// SIMATIC STEP 7 (V5.x) project Daysil_Autoclav_v4
// CPU: CPU 315-2 PN/DP
// station: P_ADR_BUS
// station: Hardware
// station: SLIO_CPU_015
// program: S7 Program(1)
// program: Backup_11012025
// program: Backup_PID_11012025
// program: Backup_08032025

SYMBOL_TABLE
"AI-SENSOR-DATA"	DB 1	DB 1
"ORTAK_DATA"	DB 2	DB 2	// Ortak Veriler
"TIME_OTO_1_DB"	DB 5	SFB 4
"TIME_OTO_2_DB"	DB 6	SFB 4
"TIME_OTO_1_PROSES_DB"	DB 7	SFB 4
"TIME_OTO_2_PROSES_DB"	DB 8	SFB 4
"SURELER_DB"	DB 14	FB 3
"SAFETY_DB"	DB 15	FB 2
"KAZAN1_DATA"	DB 17	DB 17
"KAZAN2_DATA"	DB 18	DB 18	// KAZAN 2 BILGILERI
"JEN1_DATA"	DB 19	DB 19
"JEN2_DATA"	DB 20	DB 20
"JEN1_PID_DATA"	DB 21	DB 21
"JEN2_PID_DATA"	DB 22	DB 22
"KAZAN1_PID_DATA"	DB 23	DB 23	// KAZAN 1 PID BILGILERI
"KAZAN2_PID_DATA"	DB 24	DB 24	// KAZAN 2 PID BILGILERI
"JEN2_KONTROL_BLOGU_DB"	DB 51	FB 50
"JEN_1_PID_DB"	DB 69	FB 58
"JEN_2_PID_DB"	DB 70	FB 58
"OTOKLAV_1_DB"	DB 94	FB 94
"OTOKLAV_2_DB"	DB 95	FB 95
"FB98_DB"	DB 98	FB 98
"FB99_DB"	DB 99	FB 99
"HMI_DATA"	DB 100	DB 100	// Hmi arayuz verileri
"KAZAN_1_PID_DB"	DB 130	FB 58
"KAZAN_2_PID_DATA"	DB 231	FB 58
"MAINBLOCK"	FB 1	FB 1	// ANA PROGRAM BLOGU
"SAFETY"	FB 2	FB 2
"SURELER"	FB 3	FB 3
"TEST_BLOGU"	FB 5	FB 5
"KAZAN_ORTAK"	FB 20	FB 20
"KAZAN_PID_ORTAK"	FB 21	FB 21
"CONT_C"	FB 41	FB 41	// Continuous Control
"KAZAN_1_PID_KONTROL"	FB 47	FB 47
"KAZAN_2_PID_KONTROL"	FB 48	FB 48
"JEN1_PID_KONTROL"	FB 49	FB 49
"JEN2_PID_KONTROL"	FB 50	FB 50	// BUAHR JENERATÖR 2 PID
"TCONT_CP"	FB 58	FB 58	// temperature PID controller with pulse generator and self-tuning
"KAZAN_1_KONTROL"	FB 94	FB 94
"KAZAN_2_KONTROL"	FB 95	FB 95
"KAZAN1_KONTROL_BLOGU"	FB 96	FB 96
"KAZAN2_KONTROL_BLOGU"	FB 97	FB 97
"JEN1_KONTROL_BLOGU"	FB 98	FB 98
"JEN2_KONTROL_BLOGU"	FB 99	FB 99
"TIME_UNSCALE"	FC 1	FC 1
"O.Vana_AciklikHesaplama"	FC 2	FC 2	// Oransal vana aciklik orani hesaplama
"Int_To_S5Time"	FC 10	FC 10
"Int_To_Second"	FC 11	FC 11
"TIM_S5TI"	FC 40	FC 40	// IEC Time to S5 Time
"SCALE"	FC 105	FC 105	// Scaling Values
"UNSCALE"	FC 106	FC 106	// Unscaling Values
"KAZAN1_ACIL_STOP"	I 0.0	BOOL	// Acil Stop
"KAZAN1_START"	I 0.1	BOOL	// Kazan 1 Start
"KAZAN1_TRANSFER"	I 0.2	BOOL	// Kazan 1 Buhar Transferi
"KAZAN1_BOSALTIM"	I 0.3	BOOL	// Kazan 1 Bosaltim
"KAZAN1_KAPAK_SW"	I 0.4	BOOL	// Kazan 1 Kapak Kapandi
"KAZAN2_ACIL_STOP"	I 0.5	BOOL	// Kazan 2 Acil Stop
"KAZAN2_START"	I 0.6	BOOL	// Kazan 2 Start
"KAZAN2_TRANSFER"	I 0.7	BOOL	// Kazan 2 Buhar Transferi
"KAZAN2_BOSALTIM"	I 1.0	BOOL	// Kazan 2 Bosaltim
"KAZAN2_KAPAK_SW"	I 1.1	BOOL	// Kazan 2 Kapak Kapandi
"JEN1_STOP"	I 1.2	BOOL	// Jenerator 1 Stop
"JEN1_START"	I 1.3	BOOL	// Jenerator 1 Start
"JEN2_STOP"	I 1.4	BOOL	// Jenerator 2 Stop
"JEN2_START"	I 1.5	BOOL	// Jenerator 2 Start
"MANUEL"	I 1.6	BOOL	// Manuel Mod
"OTOMATIK"	I 1.7	BOOL	// Otomatik Mod
"JEN2_MOTOR_CALISTI"	I 2.0	BOOL
"JEN_1_MIN_SU_SEVIYESI"	I 3.0	BOOL
"JEN_2_MIN_SU_SEVIYESI"	I 3.1	BOOL
"0.1 SN."	M 0.0	BOOL
"0.2 SN."	M 0.1	BOOL
"0.4 SN."	M 0.2	BOOL
"0.5 SN."	M 0.3	BOOL
"0.8 SN."	M 0.4	BOOL
"1.0 SN."	M 0.5	BOOL
"1.6 SN."	M 0.6	BOOL
"2.0 SN."	M 0.7	BOOL
"Oto_1_Proses_BASLADI"	M 20.0	BOOL
"Oto_2_Proses_Basladi"	M 20.1	BOOL
"JEN2_CALIS_SURESI_BASLA"	M 22.0	BOOL
"JEN2_CALISTI_RIS"	M 22.1	BOOL
"JEN1_CALIS_SURESI_BASLA"	M 23.0	BOOL
"JEN1_CALISTI_RIS"	M 23.1	BOOL
"Jen1_Guvenlik_set_reset"	M 25.0	BOOL
"Jen2_Guvenlik_Set_Reset"	M 26.0	BOOL
"OTO_1_BEKLEME_BASLADI"	M 27.0	BOOL
"OTO_2_BEKLEME_BASLADI"	M 27.1	BOOL
"KAZAN_1_PID_MAN_ON"	M 35.0	BOOL
"KAZAN_2_MAN_ON"	M 37.0	BOOL
"TEST_START"	M 40.0	BOOL
"TEST_STOP"	M 40.1	BOOL
"TEST_OUT"	M 40.2	BOOL
"ALWAYS OFF"	M 100.0	BOOL	// ALWAYS OFF
"ALWAYS ON"	M 100.1	BOOL	// ALWAYS ON
"SET2_ULASMADI_SR"	M 101.0	BOOL
"SET2_ULASMADI_RIS"	M 101.1	BOOL
"JEN2_TCONT_MAN_ON"	M 155.0	BOOL
"Jen2_Stop_Trigger"	M 200.0	BOOL
"Jen2_Stop_Ris"	M 200.1	BOOL
"Jen2_Stop_Set_Mem"	M 200.2	BOOL
"JEN2_STOP_SET_RESET"	M 201.0	BOOL
"Sicaklik Dustu"	M 201.1	BOOL
"Ris_Jen2_Sicaklik_Dustu"	M 201.2	BOOL
"Rising_Sogutma"	M 201.3	BOOL
"Falling_Sogutma"	M 201.4	BOOL
"JEN1_STOP_SET_RESET"	M 202.0	BOOL
"START"	M 700.1	BOOL
"PID_START"	M 700.2	BOOL
"BRULOR_START"	M 700.3	BOOL
"SICAKLIK_1_OK"	M 700.5	BOOL
"SICAKLIK_2_OK"	M 700.6	BOOL
"BURLOR_MOTOR_START"	M 700.7	BOOL
"STOP"	M 701.1	BOOL
"100_DERECE_RIS"	M 750.0	BOOL
"Jen2_Ris"	M 750.4	BOOL
"Jen1_Ris"	M 750.5	BOOL
"BOS"	M 1000.0	BOOL
"O.VanaIlkAciklik"	MD 42	REAL	// Oransal vana ilk aciklik orani
"O.VanaKademeArtis"	MD 46	REAL	// Oransal vana kademeli artis orani
"PID BLOCK"	OB 35	OB 35	// PID BLOCK
"ZAMANHATASI"	OB 80	OB 80	// ZAMAN HATASI
"GERILIMHATASI"	OB 81	OB 81	// BESLEME GERILIMI HATASI
"HATAUYARISI"	OB 82	OB 82	// HATA UYARISI
"TAKMACIKARMAHATASI"	OB 83	OB 83	// TAKMA ÇIKARMA UYARISI
"CPUHARDWAREERROR"	OB 84	OB 84	// CPU HARDWARE ERROR
"PROGRAMHATASI"	OB 85	OB 85	// PROGRAM YURUTME HATASI
"RACKHATASI"	OB 86	OB 86	// RACK HATASI
"HABERLESMEHATASI"	OB 87	OB 87	// HABERLESME HATASI,
"COMPLETE RESTART"	OB 100	OB 100	// Complete Restart
"RESTART"	OB 101	OB 101	// Restart
"COLD RESTART"	OB 102	OB 102	// Cold Restart
"PROGRAMMINGERROR"	OB 121	OB 121	// PROGRAMLAMA HATASI
"MOD_ERR"	OB 122	OB 122	// Module Access Error
"KAZAN1_YESIL_LAMBA"	Q 0.0	BOOL	// Kazan 1 Yesil Lamba
"KAZAN1_KIRMIZI_LAMBA"	Q 0.1	BOOL	// Kazan 1 Kirmizi Lamba
"KAZAN1_DUDUK"	Q 0.2	BOOL	// Kazan 1 Duduk
"KAZAN1_BOSALTIM_VALFI"	Q 0.3	BOOL	// Kazan 1 Buhar Bosaltim
"KAZAN1_TRANS_BUT_LAMBASI"	Q 0.4	BOOL	// Kazan 1 Transfer Lambasi
"KAZAN1_EMN_VALFI_BOS"	Q 0.5	BOOL	// Kazan  1 Emniyet vantili bosaltim valfi
"KAZAN2_YESIL_LAMBA"	Q 0.6	BOOL	// Kazan 2 Yesil Lamba
"KAZAN2_KIRMIZI_LAMBA"	Q 0.7	BOOL	// Kazan 2 Kirmizi Lamba
"KAZAN2_DUDUK"	Q 1.0	BOOL	// Kazan 2 Duduk
"KAZAN2_BOSALTIM_VALFI"	Q 1.1	BOOL	// Kazan 2 Buhar Bosaltim
"KAZAN2_TRANS_BUT_LAMBASI"	Q 1.2	BOOL	// Kazan 2 Transfer Lambasi
"KAZAN2_EMN_VALFI_BOS"	Q 1.3	BOOL	// Kazan Emniyet vantili bosaltim valfi
"JEN_1_HAT_VANASI"	Q 1.4	BOOL
"JEN_1_PANO_STOP_LAMBASI"	Q 1.5	BOOL
"JEN_1_PANO_START_LAMBASI"	Q 1.6	BOOL
"JEN_2_HAT_VANASI"	Q 1.7	BOOL
"JEN_2_PANO_STOP_LAMBASI"	Q 2.0	BOOL
"JEN_2_PANO_START_LAMBASI"	Q 2.1	BOOL
"PANO_OTO_MAN_BUTON_LAMBA"	Q 2.2	BOOL
"PANO_ALARM"	Q 2.3	BOOL
"JEN_1_BRULOR"	Q 2.4	BOOL
"JEN_1_POMPA"	Q 2.5	BOOL
"JEN_2_BRULOR_OUT"	Q 2.6	BOOL
"JEN_2_SU_POM_OUT"	Q 2.7	BOOL
"TON"	SFB 4	SFB 4	// Generate an On Delay
"TIME_TCK"	SFC 64	SFC 64	// Read the System Time
"delay_300ms_1"	T 8	TIMER
"500ms_delay1"	T 10	TIMER
"1s Delay"	T 11	TIMER
"Pisim_Suresi"	T 12	TIMER
"500ms_delay"	T 13	TIMER
"s_offt_7s_delay"	T 14	TIMER
"tm_adim1_pid_basla_delay"	T 16	TIMER
"500ms_delay_kazan_2"	T 20	TIMER
"1ms_delay_kazan_2"	T 21	TIMER
"kazan_2_pisirme_delay"	T 22	TIMER
"kazan_2_500ms_delay"	T 23	TIMER
"kazan_2_7s_delay"	T 24	TIMER
"Delay_500ms_Jen2"	T 30	TIMER
"DELAY_1S_JEN_HATA"	T 33	TIMER
"DELAY_300MS"	T 42	TIMER
"DELAY_500MS_1"	T 43	TIMER
"DELAY_5S_pompa"	T 44	TIMER
"OTO_2_DELAY_BITIS"	T 50	TIMER
"OTO_1_DELAY_PISIM_BITTI"	T 51	TIMER
"DELAY_ADIM5_BEKLE"	T 52	TIMER
"DELAY_ADIM5_BEKLE2"	T 53	TIMER
"TIM_SET2_ULASMADI"	T 57	TIMER
"VAT_1"	VAT 1	
END_SYMBOL_TABLE

FUNCTION_BLOCK "MAINBLOCK"	// FB 1
VERSION : 0.1
BEGIN
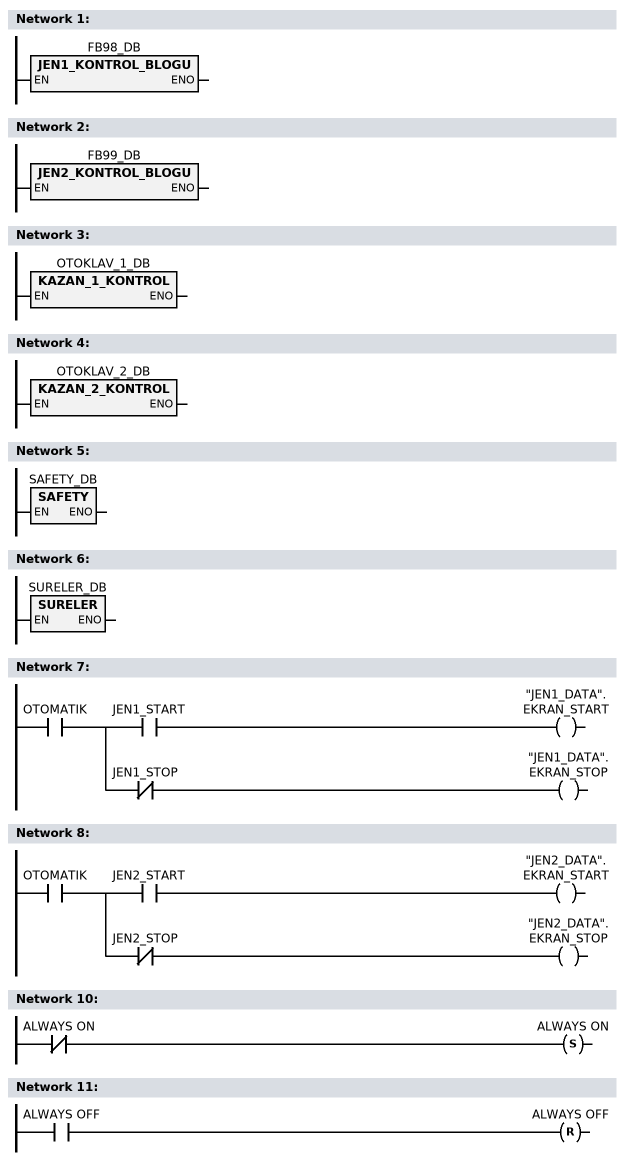
NETWORK
TITLE =
      CALL  "JEN1_KONTROL_BLOGU" , "FB98_DB";
      NOP   0;
NETWORK
TITLE =
      CALL  "JEN2_KONTROL_BLOGU" , "FB99_DB";
      NOP   0;
NETWORK
TITLE =
      CALL  "KAZAN_1_KONTROL" , "OTOKLAV_1_DB";
      NOP   0;
NETWORK
TITLE =
      CALL  "KAZAN_2_KONTROL" , "OTOKLAV_2_DB";
      NOP   0;
NETWORK
TITLE =
      CALL  "SAFETY" , "SAFETY_DB";
      NOP   0;
NETWORK
TITLE =
      CALL  "SURELER" , "SURELER_DB";
      NOP   0;
NETWORK
TITLE =
      A     "OTOMATIK";
      =     L 0.0;
      A     L 0.0;
      A     "JEN1_START";
      =     "JEN1_DATA".EKRAN_START;
      A     L 0.0;
      AN    "JEN1_STOP";
      =     "JEN1_DATA".EKRAN_STOP;
NETWORK
TITLE =
      A     "OTOMATIK";
      =     L 0.0;
      A     L 0.0;
      A     "JEN2_START";
      =     "JEN2_DATA".EKRAN_START;
      A     L 0.0;
      AN    "JEN2_STOP";
      =     "JEN2_DATA".EKRAN_STOP;
NETWORK
TITLE =
NETWORK
TITLE =
      AN    "ALWAYS ON";
      S     "ALWAYS ON";
NETWORK
TITLE =
      A     "ALWAYS OFF";
      R     "ALWAYS OFF";
NETWORK
TITLE =
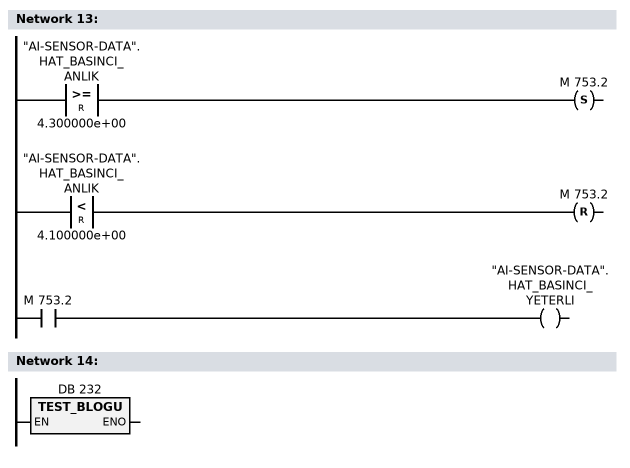
NETWORK
TITLE =
      A(;
      L     "AI-SENSOR-DATA".HAT_BASINCI_ANLIK;
      L     4.300000e+00;
      >=R;
      );
      S     M 753.2;
      A(;
      L     "AI-SENSOR-DATA".HAT_BASINCI_ANLIK;
      L     4.100000e+00;
      <R;
      );
      R     M 753.2;
      A     M 753.2;
      =     "AI-SENSOR-DATA".HAT_BASINCI_YETERLI;
NETWORK
TITLE =
      CALL  "TEST_BLOGU" , DB 232;
      NOP   0;
END_FUNCTION_BLOCK

FUNCTION_BLOCK "SAFETY"	// FB 2
VERSION : 0.1
BEGIN
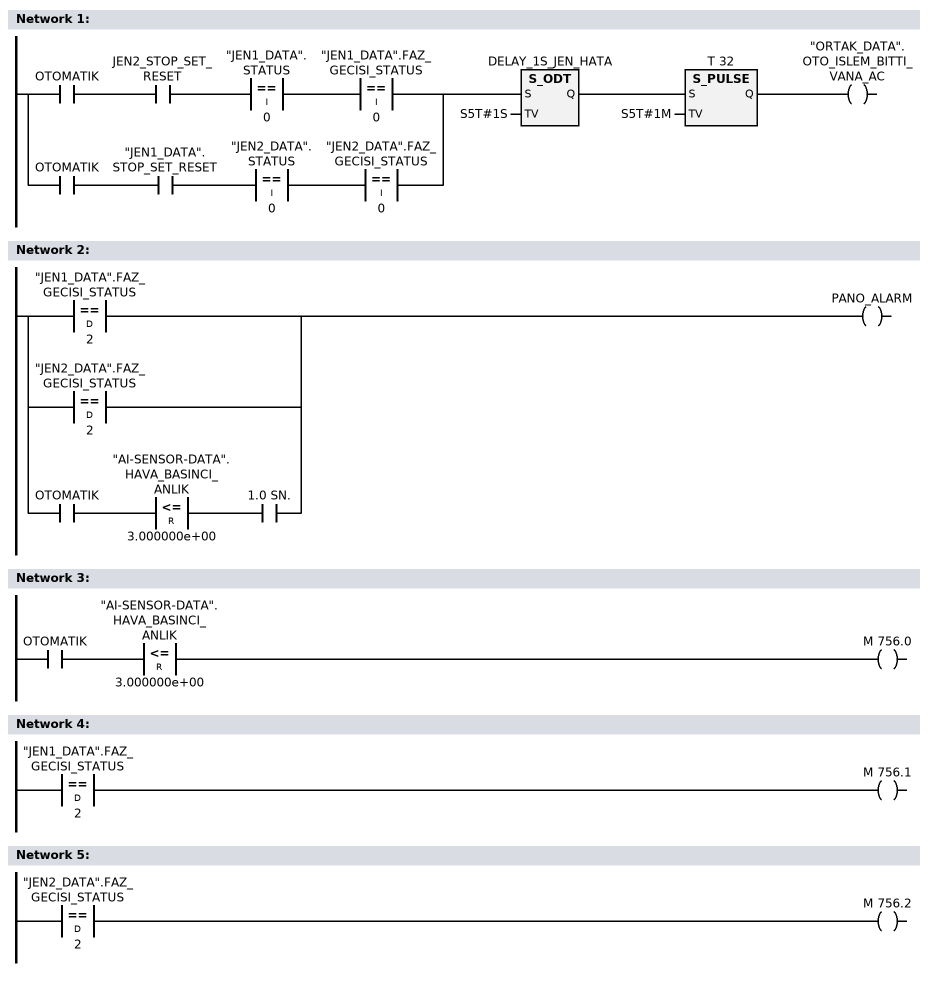
NETWORK
TITLE =
      A(;
      A(;
      A     "OTOMATIK";
      A     "JEN2_STOP_SET_RESET";
      A(;
      L     "JEN1_DATA".STATUS;
      L     0;
      ==I;
      );
      A(;
      L     "JEN1_DATA".FAZ_GECISI_STATUS;
      L     0;
      ==I;
      );
      O;
      A     "OTOMATIK";
      A     "JEN1_DATA".STOP_SET_RESET;
      A(;
      L     "JEN2_DATA".STATUS;
      L     0;
      ==I;
      );
      A(;
      L     "JEN2_DATA".FAZ_GECISI_STATUS;
      L     0;
      ==I;
      );
      );
      L     S5T#1S;
      SD    "DELAY_1S_JEN_HATA";
      NOP   0;
      NOP   0;
      NOP   0;
      A     "DELAY_1S_JEN_HATA";
      );
      L     S5T#1M;
      SP    T 32;
      NOP   0;
      NOP   0;
      NOP   0;
      A     T 32;
      =     "ORTAK_DATA".OTO_ISLEM_BITTI_VANA_AC;
NETWORK
TITLE =
      O(;
      L     "JEN1_DATA".FAZ_GECISI_STATUS;
      L     2;
      ==D;
      );
      O(;
      L     "JEN2_DATA".FAZ_GECISI_STATUS;
      L     2;
      ==D;
      );
      O;
      A     "OTOMATIK";
      A(;
      L     "AI-SENSOR-DATA".HAVA_BASINCI_ANLIK;
      L     3.000000e+00;
      <=R;
      );
      A     "1.0 SN.";
      =     "PANO_ALARM";
NETWORK
TITLE =
      A     "OTOMATIK";
      A(;
      L     "AI-SENSOR-DATA".HAVA_BASINCI_ANLIK;
      L     3.000000e+00;
      <=R;
      );
      =     M 756.0;
NETWORK
TITLE =
      L     "JEN1_DATA".FAZ_GECISI_STATUS;
      L     2;
      ==D;
      =     M 756.1;
NETWORK
TITLE =
      L     "JEN2_DATA".FAZ_GECISI_STATUS;
      L     2;
      ==D;
      =     M 756.2;
END_FUNCTION_BLOCK

FUNCTION_BLOCK "SURELER"	// FB 3
VERSION : 0.1
BEGIN
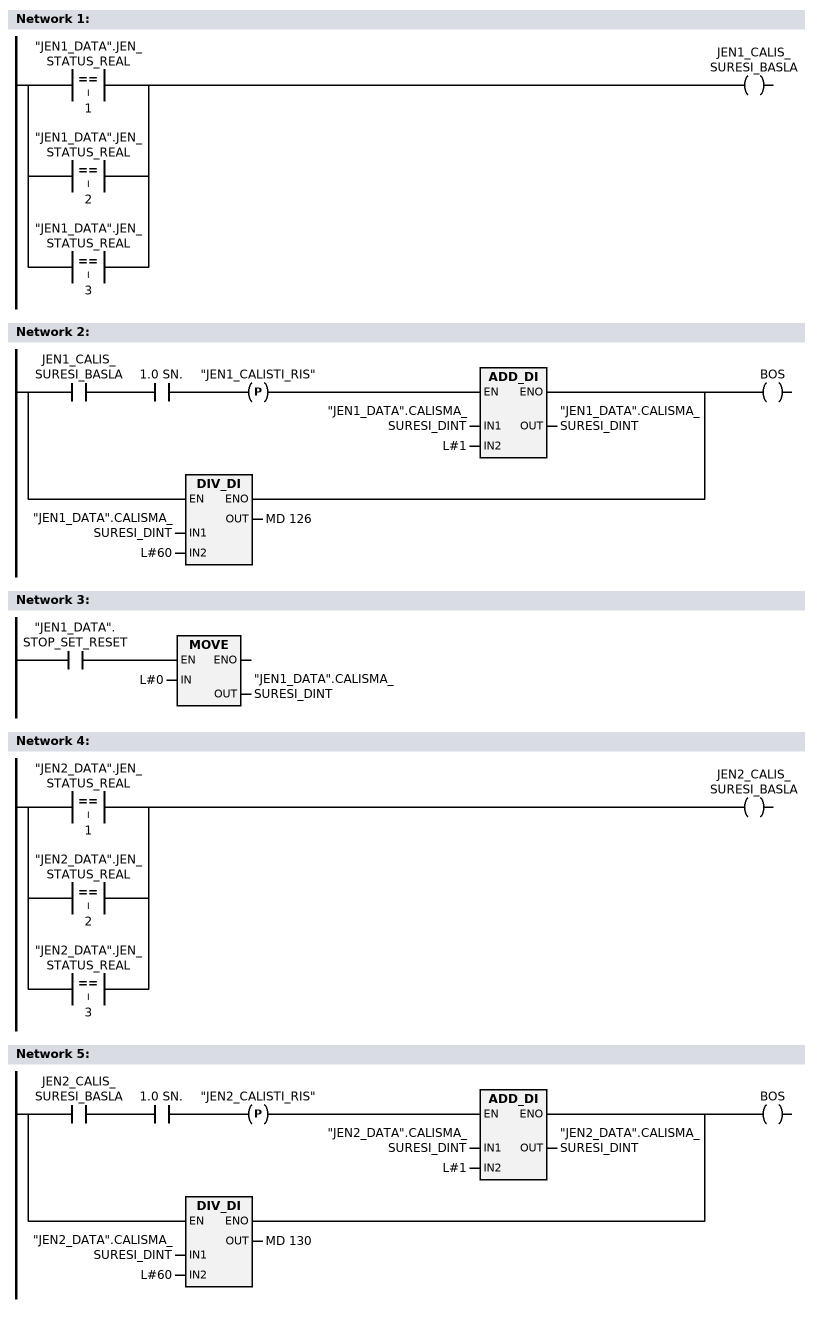
NETWORK
TITLE =
      O(;
      L     "JEN1_DATA".JEN_STATUS_REAL;
      L     1;
      ==I;
      );
      O(;
      L     "JEN1_DATA".JEN_STATUS_REAL;
      L     2;
      ==I;
      );
      O(;
      L     "JEN1_DATA".JEN_STATUS_REAL;
      L     3;
      ==I;
      );
      =     "JEN1_CALIS_SURESI_BASLA";
NETWORK
TITLE =
      O(;
      A     "JEN1_CALIS_SURESI_BASLA";
      A     "1.0 SN.";
      FP    "JEN1_CALISTI_RIS";
      JNB   _001;
      L     "JEN1_DATA".CALISMA_SURESI_DINT;
      L     L#1;
      +D;
      T     "JEN1_DATA".CALISMA_SURESI_DINT;
      AN    OV;
      SAVE;
      CLR;
_001: A     BR;
      );
      O(;
      L     "JEN1_DATA".CALISMA_SURESI_DINT;
      L     L#60;
      /D;
      T     MD 126;
      AN    OV;
      SAVE;
      CLR;
      A     BR;
      );
      =     "BOS";
NETWORK
TITLE =
      A     "JEN1_DATA".STOP_SET_RESET;
      JNB   _002;
      L     L#0;
      T     "JEN1_DATA".CALISMA_SURESI_DINT;
_002: NOP   0;
NETWORK
TITLE =
      O(;
      L     "JEN2_DATA".JEN_STATUS_REAL;
      L     1;
      ==I;
      );
      O(;
      L     "JEN2_DATA".JEN_STATUS_REAL;
      L     2;
      ==I;
      );
      O(;
      L     "JEN2_DATA".JEN_STATUS_REAL;
      L     3;
      ==I;
      );
      =     "JEN2_CALIS_SURESI_BASLA";
NETWORK
TITLE =
      O(;
      A     "JEN2_CALIS_SURESI_BASLA";
      A     "1.0 SN.";
      FP    "JEN2_CALISTI_RIS";
      JNB   _003;
      L     "JEN2_DATA".CALISMA_SURESI_DINT;
      L     L#1;
      +D;
      T     "JEN2_DATA".CALISMA_SURESI_DINT;
      AN    OV;
      SAVE;
      CLR;
_003: A     BR;
      );
      O(;
      L     "JEN2_DATA".CALISMA_SURESI_DINT;
      L     L#60;
      /D;
      T     MD 130;
      AN    OV;
      SAVE;
      CLR;
      A     BR;
      );
      =     "BOS";
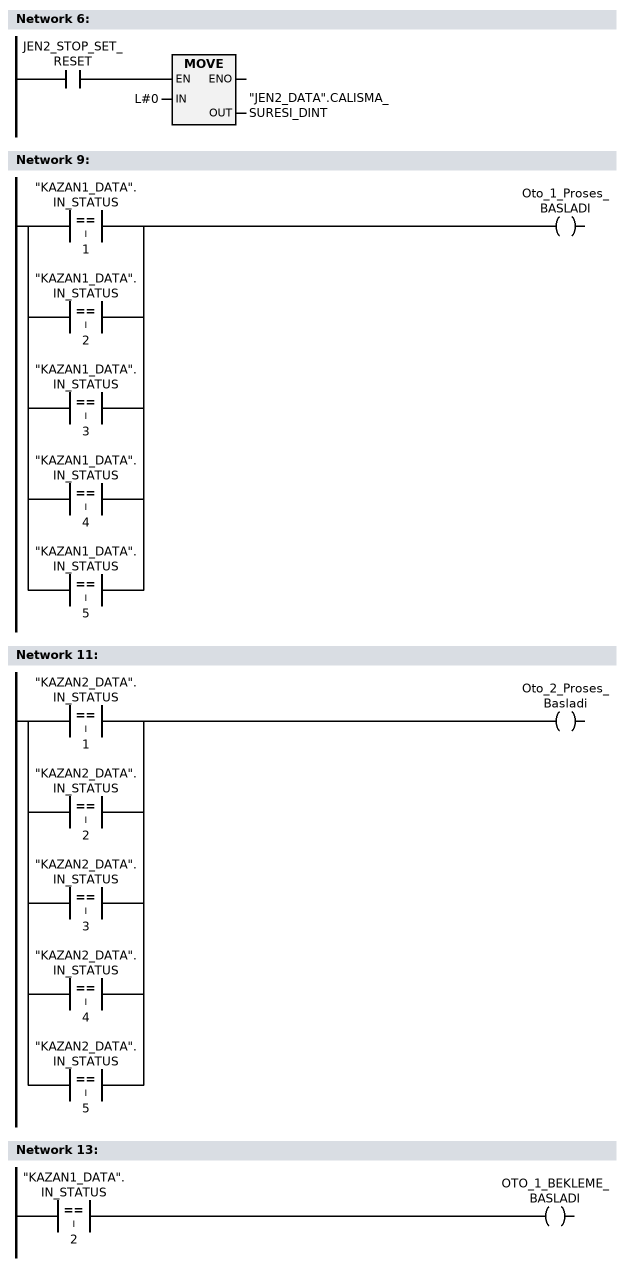
NETWORK
TITLE =
      A     "JEN2_STOP_SET_RESET";
      JNB   _004;
      L     L#0;
      T     "JEN2_DATA".CALISMA_SURESI_DINT;
_004: NOP   0;
NETWORK
TITLE =
      O(;
      A(;
      A     "KAZAN1_DATA".O_PISIM_BASLADI;
      =     L 0.0;
      BLD   103;
      BLD   9;
      =     L 5.0;
      CDB;
      OPN   DI 5;
      TAR2  LD 1;
      A     L 0.0;
      =     DIX 0.0;
      L     L#82800000;
      T     DID 2;
      LAR2  P#DBX 0.0;
      UC    "TON";
      LAR2  LD 1;
      L     DID 8;
      OPN   DI 17;
      T     DID 42;
      OPN   DI 5;
      CDB;
      BLD   10;
      A     BR;
      );
      JNB   _005;
      CALL  "TIME_UNSCALE" (
           $1                       := "KAZAN1_DATA".PISIM_GECEN_SURE_TIME,
           $2                       := "KAZAN1_DATA".IN_PISIM_SURESI,
           $3                       := "KAZAN1_DATA".PISIM_GECEN_SURE_DINT);
_005: A     BR;
      );
      O(;
      L     "KAZAN1_DATA".PISIM_GECEN_SURE_DINT;
      L     60;
      /D;
      T     MD 118;
      AN    OV;
      SAVE;
      CLR;
      A     BR;
      );
      =     "BOS";
NETWORK
TITLE =
      O(;
      A(;
      A     "KAZAN2_DATA".O_PISIM_BASLADI;
      =     L 0.0;
      BLD   103;
      BLD   9;
      =     L 5.0;
      CDB;
      OPN   DI 6;
      TAR2  LD 1;
      A     L 0.0;
      =     DIX 0.0;
      L     L#82800000;
      T     DID 2;
      LAR2  P#DBX 0.0;
      UC    "TON";
      LAR2  LD 1;
      L     DID 8;
      OPN   DI 18;
      T     DID 42;
      OPN   DI 6;
      CDB;
      BLD   10;
      A     BR;
      );
      JNB   _006;
      CALL  "TIME_UNSCALE" (
           $1                       := "KAZAN2_DATA".PISIM_GECEN_SURE_TIME,
           $2                       := "KAZAN2_DATA".IN_PISIM_SURESI,
           $3                       := "KAZAN2_DATA".PISIM_GECEN_SURE_DINT);
_006: A     BR;
      );
      O(;
      L     "KAZAN2_DATA".PISIM_GECEN_SURE_DINT;
      L     60;
      /D;
      T     MD 122;
      AN    OV;
      SAVE;
      CLR;
      A     BR;
      );
      =     "BOS";
NETWORK
TITLE =
      O(;
      L     "KAZAN1_DATA".IN_STATUS;
      L     1;
      ==I;
      );
      O(;
      L     "KAZAN1_DATA".IN_STATUS;
      L     2;
      ==I;
      );
      O(;
      L     "KAZAN1_DATA".IN_STATUS;
      L     3;
      ==I;
      );
      O(;
      L     "KAZAN1_DATA".IN_STATUS;
      L     4;
      ==I;
      );
      O(;
      L     "KAZAN1_DATA".IN_STATUS;
      L     5;
      ==I;
      );
      =     "Oto_1_Proses_BASLADI";
NETWORK
TITLE =
      O(;
      A(;
      A     "Oto_1_Proses_BASLADI";
      =     L 0.0;
      BLD   103;
      BLD   9;
      =     L 5.0;
      CDB;
      OPN   DI 7;
      TAR2  LD 1;
      A     L 0.0;
      =     DIX 0.0;
      L     L#82800000;
      T     DID 2;
      LAR2  P#DBX 0.0;
      UC    "TON";
      LAR2  LD 1;
      L     DID 8;
      OPN   DI 17;
      T     DID 50;
      OPN   DI 7;
      CDB;
      BLD   10;
      A     BR;
      );
      JNB   _007;
      L     "KAZAN1_DATA".PROSES_SURESI_TIME;
      L     1000;
      /D;
      T     "KAZAN1_DATA".PROSES_SURESI_DINT;
      AN    OV;
      SAVE;
      CLR;
_007: A     BR;
      );
      O(;
      L     "KAZAN1_DATA".PROSES_SURESI_DINT;
      L     60;
      /D;
      T     MD 110;
      AN    OV;
      SAVE;
      CLR;
      A     BR;
      );
      =     "BOS";
NETWORK
TITLE =
      O(;
      L     "KAZAN2_DATA".IN_STATUS;
      L     1;
      ==I;
      );
      O(;
      L     "KAZAN2_DATA".IN_STATUS;
      L     2;
      ==I;
      );
      O(;
      L     "KAZAN2_DATA".IN_STATUS;
      L     3;
      ==I;
      );
      O(;
      L     "KAZAN2_DATA".IN_STATUS;
      L     4;
      ==I;
      );
      O(;
      L     "KAZAN2_DATA".IN_STATUS;
      L     5;
      ==I;
      );
      =     "Oto_2_Proses_Basladi";
NETWORK
TITLE =
      O(;
      A(;
      A     "Oto_2_Proses_Basladi";
      =     L 0.0;
      BLD   103;
      BLD   9;
      =     L 5.0;
      CDB;
      OPN   DI 8;
      TAR2  LD 1;
      A     L 0.0;
      =     DIX 0.0;
      L     L#82800000;
      T     DID 2;
      LAR2  P#DBX 0.0;
      UC    "TON";
      LAR2  LD 1;
      L     DID 8;
      OPN   DI 18;
      T     DID 50;
      OPN   DI 8;
      CDB;
      BLD   10;
      A     BR;
      );
      JNB   _008;
      L     "KAZAN2_DATA".PROSES_SURESI_TIM;
      L     1000;
      /D;
      T     "KAZAN2_DATA".PROSES_SURESI_DINT;
      AN    OV;
      SAVE;
      CLR;
_008: A     BR;
      );
      O(;
      L     "KAZAN2_DATA".PROSES_SURESI_DINT;
      L     60;
      /D;
      T     MD 114;
      AN    OV;
      SAVE;
      CLR;
      A     BR;
      );
      =     "BOS";
NETWORK
TITLE =
      L     "KAZAN1_DATA".IN_STATUS;
      L     2;
      ==I;
      =     "OTO_1_BEKLEME_BASLADI";
NETWORK
TITLE =
      A(;
      A     "OTO_1_BEKLEME_BASLADI";
      =     L 0.0;
      BLD   103;
      BLD   9;
      =     L 5.0;
      CDB;
      OPN   DI 9;
      TAR2  LD 1;
      A     L 0.0;
      =     DIX 0.0;
      L     L#82800000;
      T     DID 2;
      LAR2  P#DBX 0.0;
      UC    "TON";
      LAR2  LD 1;
      L     DID 8;
      OPN   DI 17;
      T     DID 58;
      OPN   DI 9;
      CDB;
      BLD   10;
      A     BR;
      );
      JNB   _009;
      L     "KAZAN1_DATA".BEKLEME_SURESI_TIME;
      L     1000;
      /D;
      T     "KAZAN1_DATA".BEKLEME_SURESI_DINT;
_009: NOP   0;
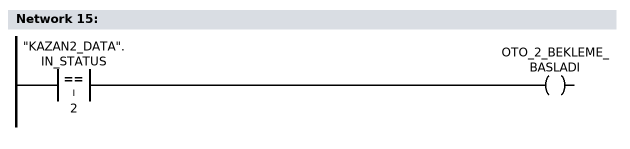
NETWORK
TITLE =
      L     "KAZAN2_DATA".IN_STATUS;
      L     2;
      ==I;
      =     "OTO_2_BEKLEME_BASLADI";
NETWORK
TITLE =
      A(;
      A     "OTO_2_BEKLEME_BASLADI";
      =     L 0.0;
      BLD   103;
      BLD   9;
      =     L 5.0;
      CDB;
      OPN   DI 10;
      TAR2  LD 1;
      A     L 0.0;
      =     DIX 0.0;
      L     L#82800000;
      T     DID 2;
      LAR2  P#DBX 0.0;
      UC    "TON";
      LAR2  LD 1;
      L     DID 8;
      OPN   DI 18;
      T     DID 58;
      OPN   DI 10;
      CDB;
      BLD   10;
      A     BR;
      );
      JNB   _00a;
      L     "KAZAN2_DATA".BEKLEME_SURESI_TIME;
      L     1000;
      /D;
      T     "KAZAN2_DATA".BEKLEME_SURESI_DINT;
_00a: NOP   0;
END_FUNCTION_BLOCK

FUNCTION_BLOCK "TEST_BLOGU"	// FB 5
VERSION : 0.1
BEGIN
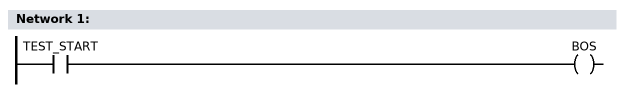
NETWORK
TITLE =
      A     "TEST_START";
      =     "BOS";
END_FUNCTION_BLOCK

FUNCTION_BLOCK "KAZAN_ORTAK"	// FB 20
VERSION : 0.1
VAR_INPUT
  IN_ACIL_STOP : BOOL ;
  IN_START : BOOL ;
  IN_TRANSFER : BOOL ;
  IN_BOSALTIM : BOOL ;
  IN_KAPAK : BOOL ;
  IN_JEN1_OK : BOOL ;
  IN_JEN2_OK : BOOL ;
  IN_JENS_OK : BOOL ;
  IN_TRANSFERE_HAZIR : BOOL ;
  IN_PISIM_SURESI : S5TIME ;
  IN_SCALE_BASINC_PER : INT ;
  IN_SET_BASINC : REAL ;
  IN_DIGER_KAZAN_BASINCI : REAL ;
  IN_TIMER_500MS : TIMER ;
  IN_TIMER_1S : TIMER ;
  IN_TIMER_PISIRME : TIMER ;
  IN_TIMER_500MS_2 : TIMER ;
  IN_TIMER_7S : TIMER ;
  IN_SCALE_HI_LIM : REAL ;
  IN_SCALE_LO_LIM : REAL ;
  IN_SCALE_SICAKLIK_HI_LIM : REAL ;
  IN_SCALE_SICAKLIK_LO_LIM : REAL ;
  IN_SCALE_SICAKLIK_PER : INT ;
  IN_DIGER_KAZAN_BOSALTIMD : BOOL ;
  IN_TRANSFER_BASLADI : BOOL ;
  IN_PISIM_SURESI_TIME_DB : BLOCK_DB ;
  IN_DIG_KAZAN_PROSES_BAS : BOOL ;
  IN_JEN_DURDU : BOOL ;
  IN_JEN_DURDUR_PID_MAN : REAL ;
  IN_DELAY_BITISI_BEKLE : TIMER ;
  IN_DELAY_BIRAZ_BEKLE : TIMER ;
  IN31 : TIMER ;
  IN32 : TIMER ;
  Bos_Vana_Period_Timer : TIMER ;
  Bos_Vana_Aciklik_Timer : TIMER ;
  BosVana_Per_TimeInterval : INT ;	//Bosaltim vanasi periyod timer interval degeri
  BosVana_Aci_TimeInterval : INT ;	//Bosaltim vanasi aciklik timer interval degeri
  BosVana_Acik_Sayisi : INT ;	//Bosaltim valfi acik kalma tekrar sayisi
END_VAR
VAR_OUTPUT
  O_YESIL_LAM : BOOL ;
  O_KIRMIZI_LAM : BOOL ;
  O_DUDUK : BOOL ;
  O_BOSALTIM_VALFI : BOOL ;
  O_PID_MAN_ON : BOOL ;
  O_PID_MAN : REAL ;
  O_TRANSFER_YAPILIYOR : BOOL ;
  O_SCALE_BASINC_RET_VAL : WORD ;
  O_SCALE_BASINC_OUT : REAL ;
  O_EMNIYET_VALFI : BOOL ;
  O_TRANSFERE_HAZIR : BOOL ;
  O_SCALE_SICAKLIK_RET_VAL : WORD ;
  O_SCALE_SICAKLIK_OUT : REAL ;
  O_TRANSFER_ET_LAMBASI : BOOL ;
  O_PROSES_BASLADI : BOOL ;
  O_KAZAN_BOSALTIMDA : BOOL ;
  O_PISIM_BASLADI : BOOL ;
END_VAR
VAR_IN_OUT
  STATUS : INT ;
END_VAR
VAR
  ST_STATUS : INT ;
  ST_OUT_BOSALTIM_MEM : BOOL ;
  ST_OUT_PID_MAN_ON : BOOL ;
  ST_OUT_PID_MAN : REAL ;
  st_ris_pid_zero : BOOL ;
  st_scale_hi_lim : REAL  := 1.000000e+001;
  st_scale_lo_lim : REAL ;
  st_basinc_ok_sure_basla : BOOL ;
  st_tolerans_mul : REAL ;
  st_toleransli_basinc : REAL ;
  st_adim4_bosaltim_valfi : BOOL ;
  st_OUT_adim4_emnyet_val : BOOL ;
  st_pid_basla : BOOL ;
  st_bosalti_valfi_acil : BOOL ;
  st_scale_basinc_ret_val : WORD ;
  st_scale_basinc_out : REAL ;
  st_scale_sicaklik_ret_va : WORD ;
  st_scale_sicaklik_out : REAL ;
  ST_PROSES_BASLADI : BOOL ;
  ST_KAZAN_BOSALTIMDA : BOOL ;
  ST_BOS : BOOL ;
  ST_SET_ADD_BASINC_02 : REAL ;
  ST_GECEN_PISIM_SURESI : TIME ;
  st_5_bar_ustu : BOOL ;
  st_5_bar_alti : BOOL ;
  st_5_bar_guvenlik_SR : BOOL ;
  st_5_bar_guvenlik_mem : BOOL ;
  STAT78 : BOOL ;
  stBasVana_Per_TimeIn : S5TIME ;
  stBasVana_Aci_TimeIn : S5TIME ;
  stBasVana_Aci_Ris : BOOL ;
  stBasVana_Aci_Sayisi : INT ;
  stBosVanasini_Ac : BOOL ;
END_VAR
VAR_TEMP
  tKademe : STRUCT
   Bir : REAL ;
   Iki : REAL ;
   Uc : REAL ;
   Dort : REAL ;
   Bes : REAL ;
   Alti : REAL ;
   Yedi : REAL ;
  END_STRUCT ;
END_VAR
BEGIN
NETWORK
TITLE = BASLANGIC SARTLARI
      A(;
      A(;
      A     "ALWAYS OFF";
      =     L 28.0;
      BLD   103;
      CALL  "SCALE" (
           $1                       := #IN_SCALE_BASINC_PER,
           $2                       := #IN_SCALE_HI_LIM,
           $3                       := #IN_SCALE_LO_LIM,
           $4                       := L 28.0,
           $5                       := #st_scale_basinc_ret_val,
           $6                       := #st_scale_basinc_out);
      A     BR;
      );
      JNB   _001;
      L     #st_scale_basinc_ret_val;
      T     #O_SCALE_BASINC_RET_VAL;
      SET;
      SAVE;
      CLR;
_001: A     BR;
      );
      JNB   _002;
      L     #st_scale_basinc_out;
      T     #O_SCALE_BASINC_OUT;
_002: NOP   0;
NETWORK
TITLE =
      A(;
      A(;
      A     "ALWAYS OFF";
      =     L 28.0;
      BLD   103;
      CALL  "SCALE" (
           $1                       := #IN_SCALE_SICAKLIK_PER,
           $2                       := #IN_SCALE_SICAKLIK_HI_LIM,
           $3                       := #IN_SCALE_SICAKLIK_LO_LIM,
           $4                       := L 28.0,
           $5                       := #st_scale_sicaklik_ret_va,
           $6                       := #st_scale_sicaklik_out);
      A     BR;
      );
      JNB   _003;
      L     #st_scale_sicaklik_ret_va;
      T     #O_SCALE_SICAKLIK_RET_VAL;
      SET;
      SAVE;
      CLR;
_003: A     BR;
      );
      JNB   _004;
      L     #st_scale_sicaklik_out;
      T     #O_SCALE_SICAKLIK_OUT;
_004: NOP   0;
NETWORK
TITLE = START
      A(;
      A     "OTOMATIK";
      A     #IN_ACIL_STOP;
      A     "AI-SENSOR-DATA".HAT_BASINCI_YETERLI;
      L     S5T#200MS;
      T     LD 28;
      TAK;
      T     LD 32;
      L     #IN_TIMER_500MS;
      T     LW 36;
      L     LD 32;
      L     LD 28;
      SD    T [LW 36];
      NOP   0;
      NOP   0;
      NOP   0;
      T     LD 28;
      TAK;
      T     LD 32;
      L     #IN_TIMER_500MS;
      T     LW 36;
      L     LD 32;
      L     LD 28;
      A     T [LW 36];
      );
      A     #IN_KAPAK;
      A     #IN_START;
      A(;
      L     #STATUS;
      L     0;
      ==I;
      );
      JNB   _005;
      L     1;
      T     #STATUS;
      SET;
      SAVE;
      CLR;
_005: A     BR;
      S     #ST_PROSES_BASLADI;
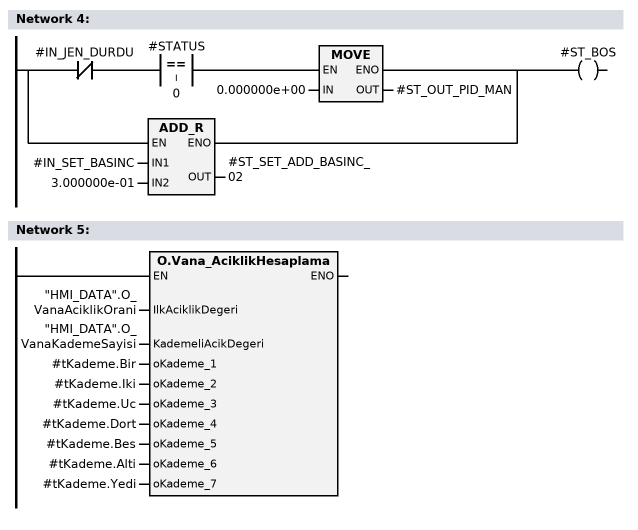
NETWORK
TITLE =
//1-Baslangicta vakum olmamasi icin bosaltim valfini ac
//Valf Normalde acik gibi dusundum
//2-Oransal valfi kapali tut
      O(;
      AN    #IN_JEN_DURDU;
      A(;
      L     #STATUS;
      L     0;
      ==I;
      );
      JNB   _006;
      L     0.000000e+00;
      T     #ST_OUT_PID_MAN;
      SET;
      SAVE;
      CLR;
_006: A     BR;
      );
      O(;
      L     #IN_SET_BASINC;
      L     3.000000e-01;
      +R;
      T     #ST_SET_ADD_BASINC_02;
      AN    OV;
      SAVE;
      CLR;
      A     BR;
      );
      =     #ST_BOS;
NETWORK
TITLE =
      CALL  "O.Vana_AciklikHesaplama" (
           IlkAciklikDegeri         := "HMI_DATA".O_VanaAciklikOrani,
           KademeliAcikDegeri       := "HMI_DATA".O_VanaKademeSayisi,
           oKademe_1                := #tKademe.Bir,
           oKademe_2                := #tKademe.Iki,
           oKademe_3                := #tKademe.Uc,
           oKademe_4                := #tKademe.Dort,
           oKademe_5                := #tKademe.Bes,
           oKademe_6                := #tKademe.Alti,
           oKademe_7                := #tKademe.Yedi);
      NOP   0;
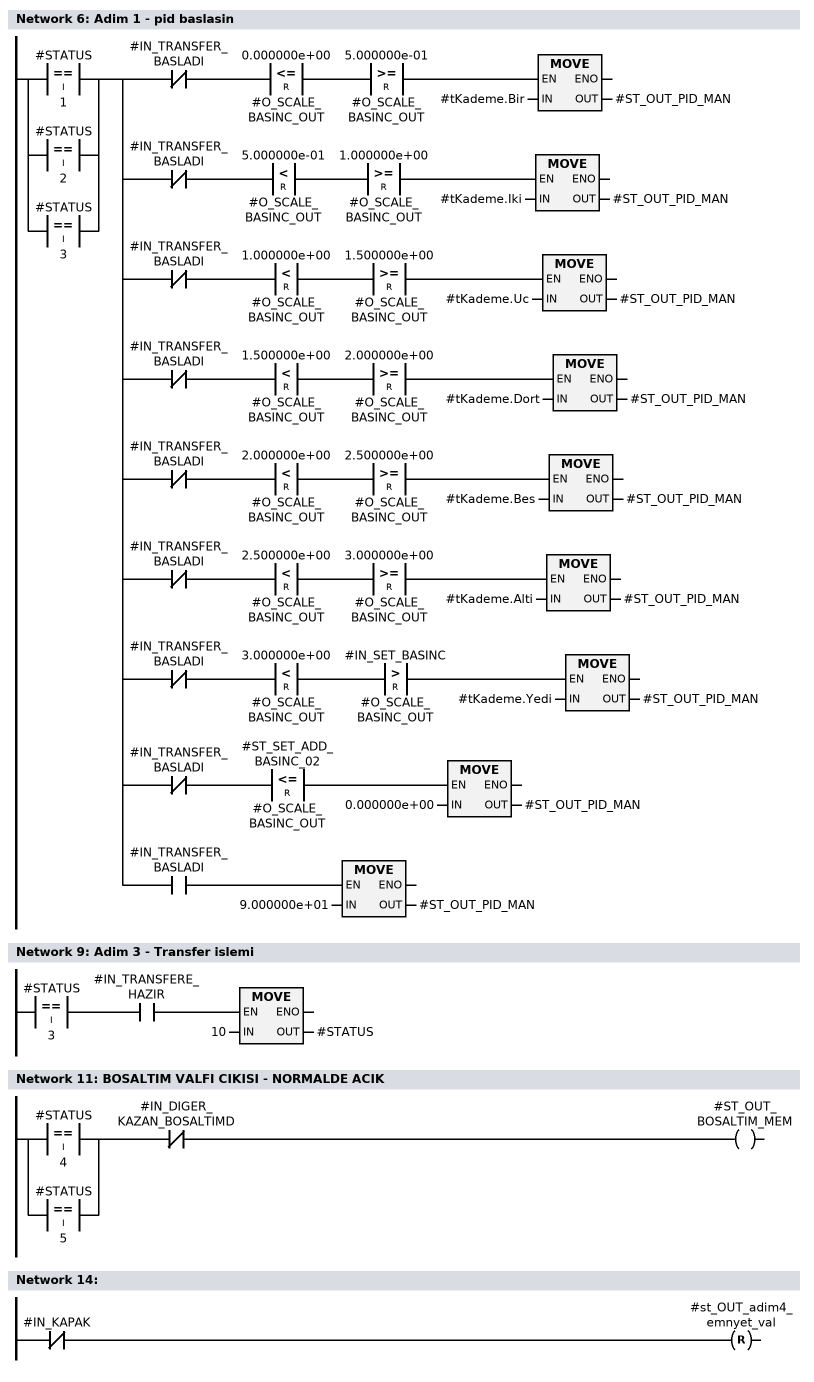
NETWORK
TITLE = Adim 1 - pid baslasin
      O(;
      L     #STATUS;
      L     1;
      ==I;
      );
      O(;
      L     #STATUS;
      L     2;
      ==I;
      );
      O(;
      L     #STATUS;
      L     3;
      ==I;
      );
      =     L 28.0;
      A     L 28.0;
      AN    #IN_TRANSFER_BASLADI;
      A(;
      L     0.000000e+00;
      L     #O_SCALE_BASINC_OUT;
      <=R;
      );
      A(;
      L     5.000000e-01;
      L     #O_SCALE_BASINC_OUT;
      >=R;
      );
      JNB   _007;
      L     #tKademe.Bir;
      T     #ST_OUT_PID_MAN;
_007: NOP   0;
      A     L 28.0;
      AN    #IN_TRANSFER_BASLADI;
      A(;
      L     5.000000e-01;
      L     #O_SCALE_BASINC_OUT;
      <R;
      );
      A(;
      L     1.000000e+00;
      L     #O_SCALE_BASINC_OUT;
      >=R;
      );
      JNB   _008;
      L     #tKademe.Iki;
      T     #ST_OUT_PID_MAN;
_008: NOP   0;
      A     L 28.0;
      AN    #IN_TRANSFER_BASLADI;
      A(;
      L     1.000000e+00;
      L     #O_SCALE_BASINC_OUT;
      <R;
      );
      A(;
      L     1.500000e+00;
      L     #O_SCALE_BASINC_OUT;
      >=R;
      );
      JNB   _009;
      L     #tKademe.Uc;
      T     #ST_OUT_PID_MAN;
_009: NOP   0;
      A     L 28.0;
      AN    #IN_TRANSFER_BASLADI;
      A(;
      L     1.500000e+00;
      L     #O_SCALE_BASINC_OUT;
      <R;
      );
      A(;
      L     2.000000e+00;
      L     #O_SCALE_BASINC_OUT;
      >=R;
      );
      JNB   _00a;
      L     #tKademe.Dort;
      T     #ST_OUT_PID_MAN;
_00a: NOP   0;
      A     L 28.0;
      AN    #IN_TRANSFER_BASLADI;
      A(;
      L     2.000000e+00;
      L     #O_SCALE_BASINC_OUT;
      <R;
      );
      A(;
      L     2.500000e+00;
      L     #O_SCALE_BASINC_OUT;
      >=R;
      );
      JNB   _00b;
      L     #tKademe.Bes;
      T     #ST_OUT_PID_MAN;
_00b: NOP   0;
      A     L 28.0;
      AN    #IN_TRANSFER_BASLADI;
      A(;
      L     2.500000e+00;
      L     #O_SCALE_BASINC_OUT;
      <R;
      );
      A(;
      L     3.000000e+00;
      L     #O_SCALE_BASINC_OUT;
      >=R;
      );
      JNB   _00c;
      L     #tKademe.Alti;
      T     #ST_OUT_PID_MAN;
_00c: NOP   0;
      A     L 28.0;
      AN    #IN_TRANSFER_BASLADI;
      A(;
      L     3.000000e+00;
      L     #O_SCALE_BASINC_OUT;
      <R;
      );
      A(;
      L     #IN_SET_BASINC;
      L     #O_SCALE_BASINC_OUT;
      >R;
      );
      JNB   _00d;
      L     #tKademe.Yedi;
      T     #ST_OUT_PID_MAN;
_00d: NOP   0;
      A     L 28.0;
      AN    #IN_TRANSFER_BASLADI;
      A(;
      L     #ST_SET_ADD_BASINC_02;
      L     #O_SCALE_BASINC_OUT;
      <=R;
      );
      JNB   _00e;
      L     0.000000e+00;
      T     #ST_OUT_PID_MAN;
_00e: NOP   0;
      A     L 28.0;
      A     #IN_TRANSFER_BASLADI;
      JNB   _00f;
      L     9.000000e+01;
      T     #ST_OUT_PID_MAN;
_00f: NOP   0;
NETWORK
TITLE = Adim 1 - Pisim Süresi
      L     #STATUS;
      L     1;
      ==I;
      =     L 28.0;
      A(;
      A     L 28.0;
      A     #st_basinc_ok_sure_basla;
      L     #IN_PISIM_SURESI;
      T     LD 29;
      TAK;
      T     LD 33;
      L     #IN_TIMER_PISIRME;
      T     LW 37;
      L     LD 33;
      L     LD 29;
      SD    T [LW 37];
      NOP   0;
      NOP   0;
      NOP   0;
      T     LD 29;
      TAK;
      T     LD 33;
      L     #IN_TIMER_PISIRME;
      T     LW 37;
      L     LD 33;
      L     LD 29;
      A     T [LW 37];
      );
      JNB   _010;
      L     2;
      T     #STATUS;
_010: NOP   0;
      A     L 28.0;
      A(;
      O(;
      L     #O_SCALE_BASINC_OUT;
      L     #IN_SET_BASINC;
      >=R;
      );
      O     #st_basinc_ok_sure_basla;
      );
      =     #st_basinc_ok_sure_basla;
NETWORK
TITLE = ADIM 2 - Transfer yada bosaltim bekle
      L     #STATUS;
      L     2;
      ==I;
      =     L 28.0;
      A     L 28.0;
      L     S5T#5M;
      T     LD 29;
      TAK;
      T     LD 33;
      L     #IN31;
      T     LW 37;
      L     LD 33;
      L     LD 29;
      SD    T [LW 37];
      NOP   0;
      NOP   0;
      NOP   0;
      NOP   0;
      A     L 28.0;
      A     #IN_TRANSFER;
      JNB   _011;
      L     3;
      T     #STATUS;
_011: NOP   0;
      A     L 28.0;
      A     #IN_BOSALTIM;
      JNB   _012;
      L     4;
      T     #STATUS;
_012: NOP   0;
NETWORK
TITLE = Adim 3 - Transfer islemi
      A(;
      L     #STATUS;
      L     3;
      ==I;
      );
      A     #IN_TRANSFERE_HAZIR;
      JNB   _013;
      L     10;
      T     #STATUS;
_013: NOP   0;
NETWORK
TITLE = Adim 3 - Transfer islemi
      L     #STATUS;
      L     10;
      ==I;
      =     L 28.0;
      A     L 28.0;
      JNB   _014;
      L     9.000000e+01;
      T     #ST_OUT_PID_MAN;
      SET;
      SAVE;
      CLR;
_014: A     BR;
      =     #O_TRANSFER_YAPILIYOR;
      A(;
      A     L 28.0;
      L     S5T#23S;
      T     LD 29;
      TAK;
      T     LD 33;
      L     #IN_TIMER_500MS_2;
      T     LW 37;
      L     LD 33;
      L     LD 29;
      SD    T [LW 37];
      NOP   0;
      NOP   0;
      NOP   0;
      T     LD 29;
      TAK;
      T     LD 33;
      L     #IN_TIMER_500MS_2;
      T     LW 37;
      L     LD 33;
      L     LD 29;
      A     T [LW 37];
      );
      JNB   _015;
      L     4;
      T     #STATUS;
_015: NOP   0;
NETWORK
TITLE = BOSALTIM VALFI CIKISI - NORMALDE ACIK
      A(;
      O(;
      L     #STATUS;
      L     4;
      ==I;
      );
      O(;
      L     #STATUS;
      L     5;
      ==I;
      );
      );
      AN    #IN_DIGER_KAZAN_BOSALTIMD;
      =     #ST_OUT_BOSALTIM_MEM;
NETWORK
TITLE = Adim 4 - Bosaltim Adimi
      L     #STATUS;
      L     4;
      ==I;
      =     L 28.0;
      A     L 28.0;
      JNB   _016;
      L     0.000000e+00;
      T     #ST_OUT_PID_MAN;
_016: NOP   0;
      A     L 28.0;
      BLD   102;
      =     #ST_KAZAN_BOSALTIMDA;
      A     L 28.0;
      A(;
      L     #O_SCALE_BASINC_OUT;
      L     "HMI_DATA".BosIsl_BosVana_Basinc;
      <=R;
      );
      =     L 28.1;
      A     L 28.1;
      BLD   102;
      S     #st_OUT_adim4_emnyet_val;
      A(;
      A     L 28.1;
      A(;
      L     #O_SCALE_BASINC_OUT;
      L     1.000000e-01;
      <=R;
      );
      L     S5T#5S;
      T     LD 29;
      TAK;
      T     LD 33;
      L     #IN_DELAY_BITISI_BEKLE;
      T     LW 37;
      L     LD 33;
      L     LD 29;
      SD    T [LW 37];
      NOP   0;
      NOP   0;
      NOP   0;
      T     LD 29;
      TAK;
      T     LD 33;
      L     #IN_DELAY_BITISI_BEKLE;
      T     LW 37;
      L     LD 33;
      L     LD 29;
      A     T [LW 37];
      );
      JNB   _017;
      L     5;
      T     #STATUS;
_017: NOP   0;
NETWORK
TITLE = KAPAK AÇILMASINI BEKLE
      A(;
      A(;
      L     #STATUS;
      L     5;
      ==I;
      );
      L     S5T#1S;
      T     LD 28;
      TAK;
      T     LD 32;
      L     #IN_DELAY_BIRAZ_BEKLE;
      T     LW 36;
      L     LD 32;
      L     LD 28;
      SD    T [LW 36];
      NOP   0;
      NOP   0;
      NOP   0;
      T     LD 28;
      TAK;
      T     LD 32;
      L     #IN_DELAY_BIRAZ_BEKLE;
      T     LW 36;
      L     LD 32;
      L     LD 28;
      A     T [LW 36];
      );
      AN    #IN_KAPAK;
      JNB   _018;
      L     0;
      T     #STATUS;
_018: NOP   0;
NETWORK
TITLE =
      AN    #IN_KAPAK;
      R     #st_OUT_adim4_emnyet_val;
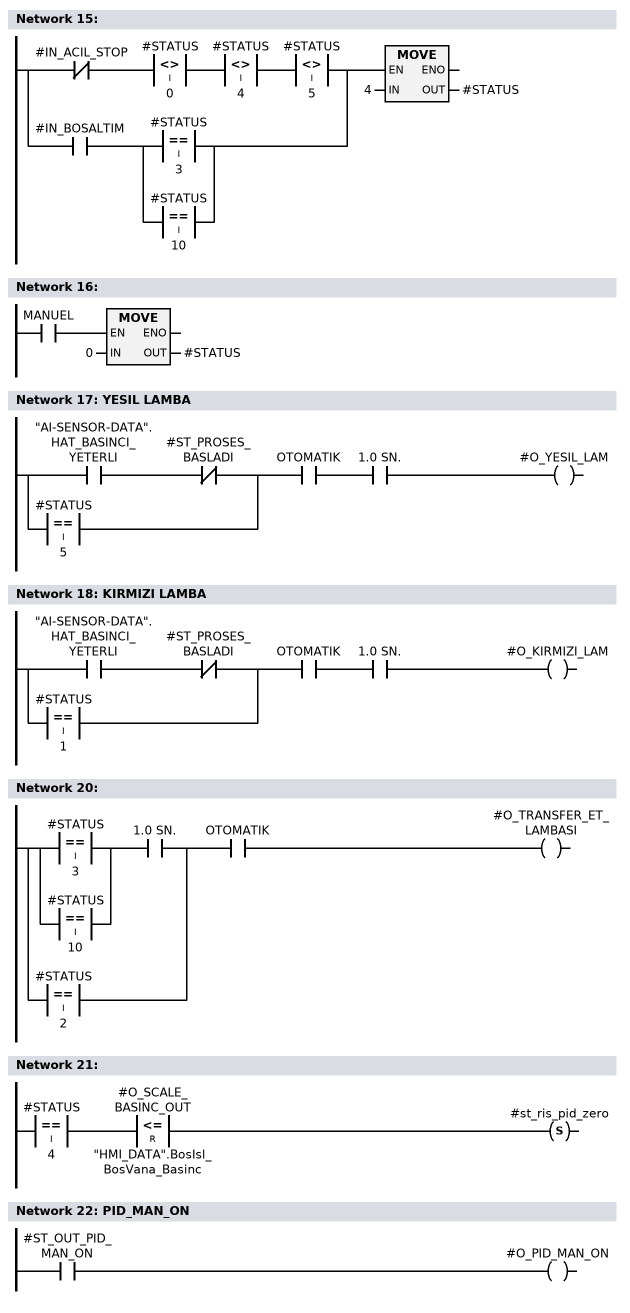
NETWORK
TITLE =
//1- Acil Stop ile 1,2 ve 3. adimda ise bosaltim adimina git 
//2- 3. adimda bosalt butonu ile bosaltim yapabilsin  
      A(;
      AN    #IN_ACIL_STOP;
      A(;
      L     #STATUS;
      L     0;
      <>I;
      );
      A(;
      L     #STATUS;
      L     4;
      <>I;
      );
      A(;
      L     #STATUS;
      L     5;
      <>I;
      );
      O;
      A     #IN_BOSALTIM;
      A(;
      O(;
      L     #STATUS;
      L     3;
      ==I;
      );
      O(;
      L     #STATUS;
      L     10;
      ==I;
      );
      );
      );
      JNB   _019;
      L     4;
      T     #STATUS;
_019: NOP   0;
NETWORK
TITLE =
      A     "MANUEL";
      JNB   _01a;
      L     0;
      T     #STATUS;
_01a: NOP   0;
NETWORK
TITLE = YESIL LAMBA
      A(;
      A     "AI-SENSOR-DATA".HAT_BASINCI_YETERLI;
      AN    #ST_PROSES_BASLADI;
      O(;
      L     #STATUS;
      L     5;
      ==I;
      );
      );
      A     "OTOMATIK";
      A     "1.0 SN.";
      =     #O_YESIL_LAM;
NETWORK
TITLE = KIRMIZI LAMBA
      A(;
      A     "AI-SENSOR-DATA".HAT_BASINCI_YETERLI;
      AN    #ST_PROSES_BASLADI;
      O(;
      L     #STATUS;
      L     1;
      ==I;
      );
      );
      A     "OTOMATIK";
      A     "1.0 SN.";
      =     #O_KIRMIZI_LAM;
NETWORK
TITLE = DUDUK
      A(;
      A(;
      L     #STATUS;
      L     2;
      ==I;
      );
      A     "1.0 SN.";
      O(;
      A(;
      O(;
      L     #STATUS;
      L     3;
      ==I;
      );
      O(;
      L     #STATUS;
      L     10;
      ==I;
      );
      );
      AN    #O_TRANSFER_YAPILIYOR;
      L     S5T#5M;
      T     LD 28;
      TAK;
      T     LD 32;
      L     #IN32;
      T     LW 36;
      L     LD 32;
      L     LD 28;
      SD    T [LW 36];
      NOP   0;
      NOP   0;
      NOP   0;
      T     LD 28;
      TAK;
      T     LD 32;
      L     #IN32;
      T     LW 36;
      L     LD 32;
      L     LD 28;
      A     T [LW 36];
      );
      );
      A     "OTOMATIK";
      =     #O_DUDUK;
NETWORK
TITLE =
      A(;
      A(;
      O(;
      L     #STATUS;
      L     3;
      ==I;
      );
      O(;
      L     #STATUS;
      L     10;
      ==I;
      );
      );
      A     "1.0 SN.";
      O(;
      L     #STATUS;
      L     2;
      ==I;
      );
      );
      A     "OTOMATIK";
      =     #O_TRANSFER_ET_LAMBASI;
NETWORK
TITLE =
      A(;
      L     #STATUS;
      L     4;
      ==I;
      );
      A(;
      L     #O_SCALE_BASINC_OUT;
      L     "HMI_DATA".BosIsl_BosVana_Basinc;
      <=R;
      );
      S     #st_ris_pid_zero;
NETWORK
TITLE = PID_MAN_ON 
      A     #ST_OUT_PID_MAN_ON;
      =     #O_PID_MAN_ON;
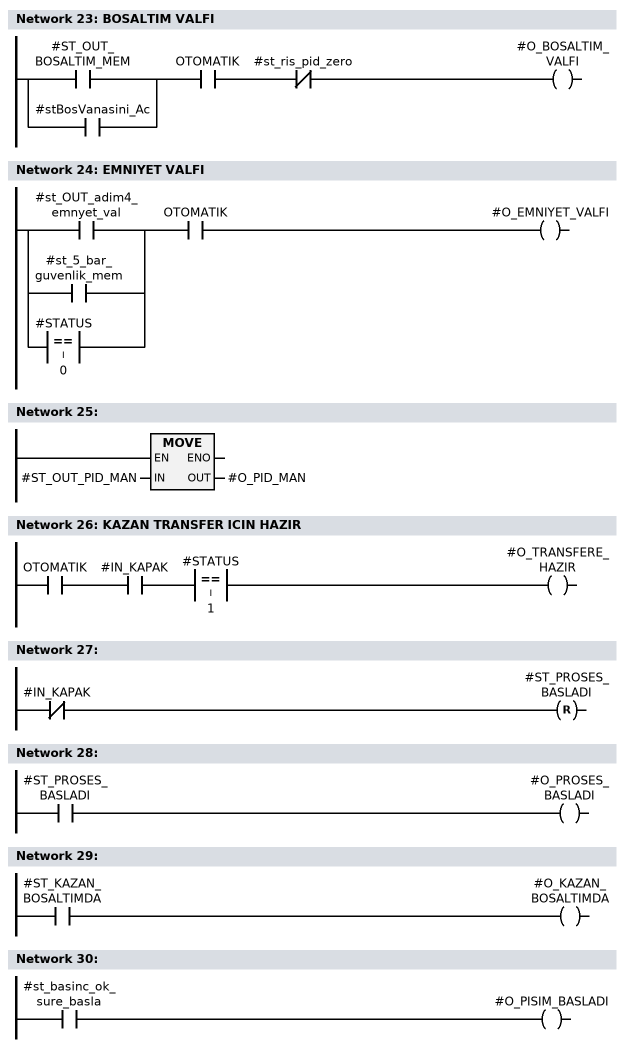
NETWORK
TITLE = BOSALTIM VALFI
      A(;
      O     #ST_OUT_BOSALTIM_MEM;
      O     #stBosVanasini_Ac;
      );
      A     "OTOMATIK";
      AN    #st_ris_pid_zero;
      =     #O_BOSALTIM_VALFI;
NETWORK
TITLE = EMNIYET VALFI
      A(;
      O     #st_OUT_adim4_emnyet_val;
      O     #st_5_bar_guvenlik_mem;
      O(;
      L     #STATUS;
      L     0;
      ==I;
      );
      );
      A     "OTOMATIK";
      =     #O_EMNIYET_VALFI;
NETWORK
TITLE =
      L     #ST_OUT_PID_MAN;
      T     #O_PID_MAN;
      NOP   0;
NETWORK
TITLE = KAZAN TRANSFER ICIN HAZIR
      A     "OTOMATIK";
      A     #IN_KAPAK;
      A(;
      L     #STATUS;
      L     1;
      ==I;
      );
      =     #O_TRANSFERE_HAZIR;
NETWORK
TITLE =
      AN    #IN_KAPAK;
      R     #ST_PROSES_BASLADI;
NETWORK
TITLE =
      A     #ST_PROSES_BASLADI;
      =     #O_PROSES_BASLADI;
NETWORK
TITLE =
      A     #ST_KAZAN_BOSALTIMDA;
      =     #O_KAZAN_BOSALTIMDA;
NETWORK
TITLE =
      A     #st_basinc_ok_sure_basla;
      =     #O_PISIM_BASLADI;
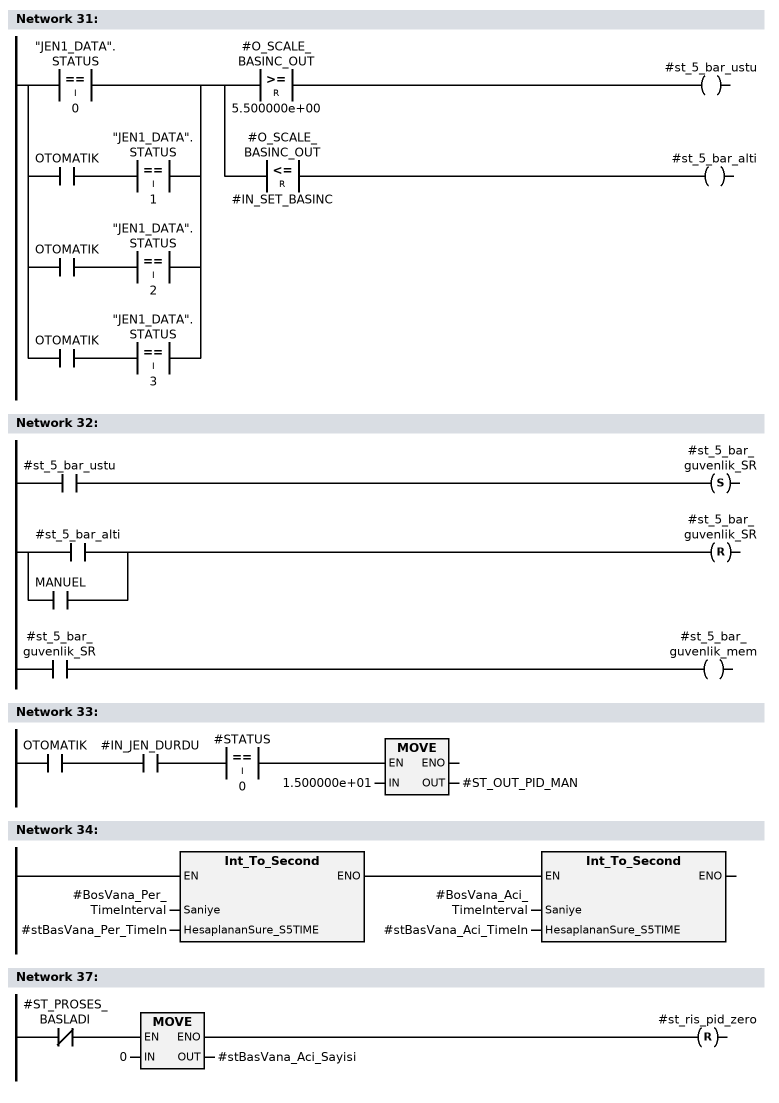
NETWORK
TITLE =
//Otoklav 5.5 bar'a geldiginde emniyet vantilini ac ve sete düþtügünde tekrar 
//emniyet ventilini kapat 
      O(;
      L     "JEN1_DATA".STATUS;
      L     0;
      ==I;
      );
      O;
      A     "OTOMATIK";
      A(;
      L     "JEN1_DATA".STATUS;
      L     1;
      ==I;
      );
      O;
      A     "OTOMATIK";
      A(;
      L     "JEN1_DATA".STATUS;
      L     2;
      ==I;
      );
      O;
      A     "OTOMATIK";
      A(;
      L     "JEN1_DATA".STATUS;
      L     3;
      ==I;
      );
      =     L 28.0;
      A     L 28.0;
      A(;
      L     #O_SCALE_BASINC_OUT;
      L     5.500000e+00;
      >=R;
      );
      =     #st_5_bar_ustu;
      A     L 28.0;
      A(;
      L     #O_SCALE_BASINC_OUT;
      L     #IN_SET_BASINC;
      <=R;
      );
      =     #st_5_bar_alti;
NETWORK
TITLE =
      A     #st_5_bar_ustu;
      S     #st_5_bar_guvenlik_SR;
      A(;
      O     #st_5_bar_alti;
      O     "MANUEL";
      );
      R     #st_5_bar_guvenlik_SR;
      A     #st_5_bar_guvenlik_SR;
      =     #st_5_bar_guvenlik_mem;
NETWORK
TITLE =
//JENERATORLER DURDUGUNDA BELIRLI SANIYE ORANSAL VANAYI AC HATTA BULUNAN BUHAR 
//TASFIYE EDILSIN
      A     "OTOMATIK";
      A     #IN_JEN_DURDU;
      A(;
      L     #STATUS;
      L     0;
      ==I;
      );
      JNB   _01b;
      L     1.500000e+01;
      T     #ST_OUT_PID_MAN;
_01b: NOP   0;
NETWORK
TITLE =
      A(;
      CALL  "Int_To_Second" (
           Saniye                   := #BosVana_Per_TimeInterval,
           HesaplananSure_S5TIME    := #stBasVana_Per_TimeIn);
      A     BR;
      );
      JNB   _01c;
      CALL  "Int_To_Second" (
           Saniye                   := #BosVana_Aci_TimeInterval,
           HesaplananSure_S5TIME    := #stBasVana_Aci_TimeIn);
_01c: NOP   0;
NETWORK
TITLE = Bosaltim vanasi periyodlu acilma islemi
      A     "OTOMATIK";
      A     #ST_PROSES_BASLADI;
      AN    #IN_DIGER_KAZAN_BOSALTIMD;
      A(;
      L     #stBasVana_Aci_Sayisi;
      L     #BosVana_Acik_Sayisi;
      <I;
      );
      =     L 28.0;
      A     L 28.0;
      T     LD 29;
      TAK;
      T     LD 33;
      L     #Bos_Vana_Aciklik_Timer;
      T     LW 37;
      L     LD 33;
      L     LD 29;
      AN    T [LW 37];
      L     #stBasVana_Per_TimeIn;
      T     LD 29;
      TAK;
      T     LD 33;
      L     #Bos_Vana_Period_Timer;
      T     LW 37;
      L     LD 33;
      L     LD 29;
      SD    T [LW 37];
      NOP   0;
      NOP   0;
      NOP   0;
      NOP   0;
      A     L 28.0;
      T     LD 29;
      TAK;
      T     LD 33;
      L     #Bos_Vana_Period_Timer;
      T     LW 37;
      L     LD 33;
      L     LD 29;
      A     T [LW 37];
      =     L 28.1;
      A     L 28.1;
      L     #stBasVana_Aci_TimeIn;
      T     LD 29;
      TAK;
      T     LD 33;
      L     #Bos_Vana_Aciklik_Timer;
      T     LW 37;
      L     LD 33;
      L     LD 29;
      SD    T [LW 37];
      NOP   0;
      NOP   0;
      NOP   0;
      NOP   0;
      A     L 28.1;
      BLD   102;
      =     #stBosVanasini_Ac;
NETWORK
TITLE =
      A     "OTOMATIK";
      T     LD 28;
      TAK;
      T     LD 32;
      L     #Bos_Vana_Period_Timer;
      T     LW 36;
      L     LD 32;
      L     LD 28;
      A     T [LW 36];
      FP    #stBasVana_Aci_Ris;
      JNB   _01d;
      L     #stBasVana_Aci_Sayisi;
      L     1;
      +I;
      T     #stBasVana_Aci_Sayisi;
_01d: NOP   0;
NETWORK
TITLE =
      AN    #ST_PROSES_BASLADI;
      JNB   _01e;
      L     0;
      T     #stBasVana_Aci_Sayisi;
      SET;
      SAVE;
      CLR;
_01e: A     BR;
      R     #st_ris_pid_zero;
END_FUNCTION_BLOCK

// FB 41: know-how protected block, not included

FUNCTION_BLOCK "KAZAN_1_PID_KONTROL"	// FB 47
VERSION : 0.1
BEGIN
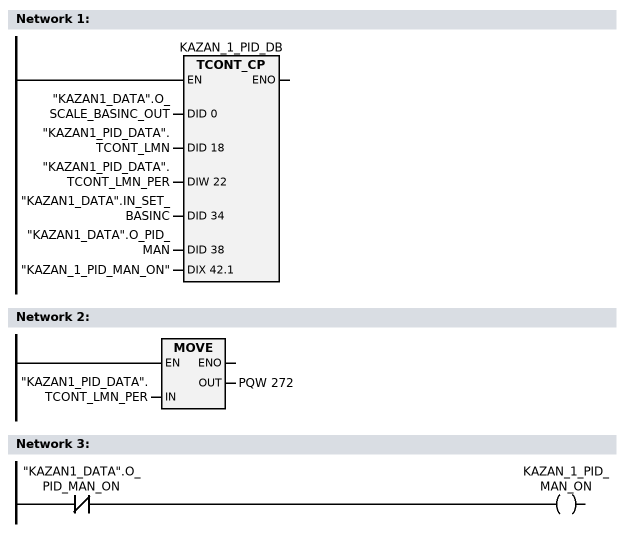
NETWORK
TITLE =
      CALL  "TCONT_CP" , "KAZAN_1_PID_DB" (
           DID 0                    := "KAZAN1_DATA".O_SCALE_BASINC_OUT,
           DID 18                   := "KAZAN1_PID_DATA".TCONT_LMN,
           DIW 22                   := "KAZAN1_PID_DATA".TCONT_LMN_PER,
           DID 34                   := "KAZAN1_DATA".IN_SET_BASINC,
           DID 38                   := "KAZAN1_DATA".O_PID_MAN,
           DIX 42.1                 := "KAZAN_1_PID_MAN_ON");
      NOP   0;
NETWORK
TITLE =
      L     "KAZAN1_PID_DATA".TCONT_LMN_PER;
      T     PQW 272;
      NOP   0;
NETWORK
TITLE =
      AN    "KAZAN1_DATA".O_PID_MAN_ON;
      =     "KAZAN_1_PID_MAN_ON";
NETWORK
TITLE =
END_FUNCTION_BLOCK

FUNCTION_BLOCK "KAZAN_2_PID_KONTROL"	// FB 48
VERSION : 0.1
BEGIN
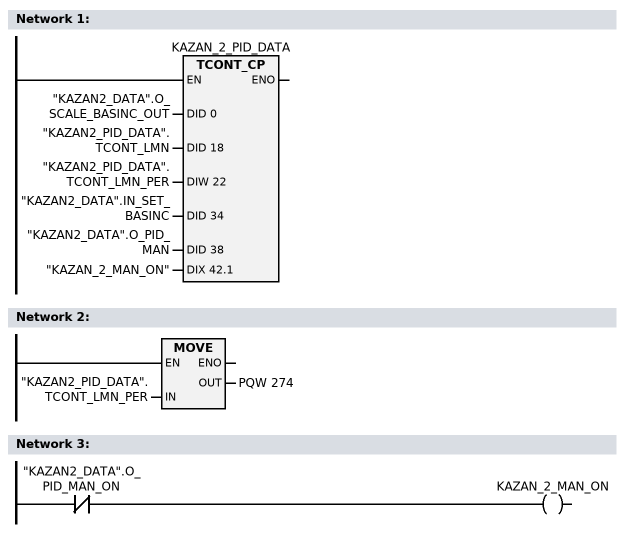
NETWORK
TITLE =
      CALL  "TCONT_CP" , "KAZAN_2_PID_DATA" (
           DID 0                    := "KAZAN2_DATA".O_SCALE_BASINC_OUT,
           DID 18                   := "KAZAN2_PID_DATA".TCONT_LMN,
           DIW 22                   := "KAZAN2_PID_DATA".TCONT_LMN_PER,
           DID 34                   := "KAZAN2_DATA".IN_SET_BASINC,
           DID 38                   := "KAZAN2_DATA".O_PID_MAN,
           DIX 42.1                 := "KAZAN_2_MAN_ON");
      NOP   0;
NETWORK
TITLE =
      L     "KAZAN2_PID_DATA".TCONT_LMN_PER;
      T     PQW 274;
      NOP   0;
NETWORK
TITLE =
      AN    "KAZAN2_DATA".O_PID_MAN_ON;
      =     "KAZAN_2_MAN_ON";
END_FUNCTION_BLOCK

FUNCTION_BLOCK "JEN1_PID_KONTROL"	// FB 49
VERSION : 0.1
VAR
  STAT0 : REAL ;
  STAT1 : BOOL ;
  STAT2 : REAL ;
  STAT3 : INT ;
END_VAR
BEGIN
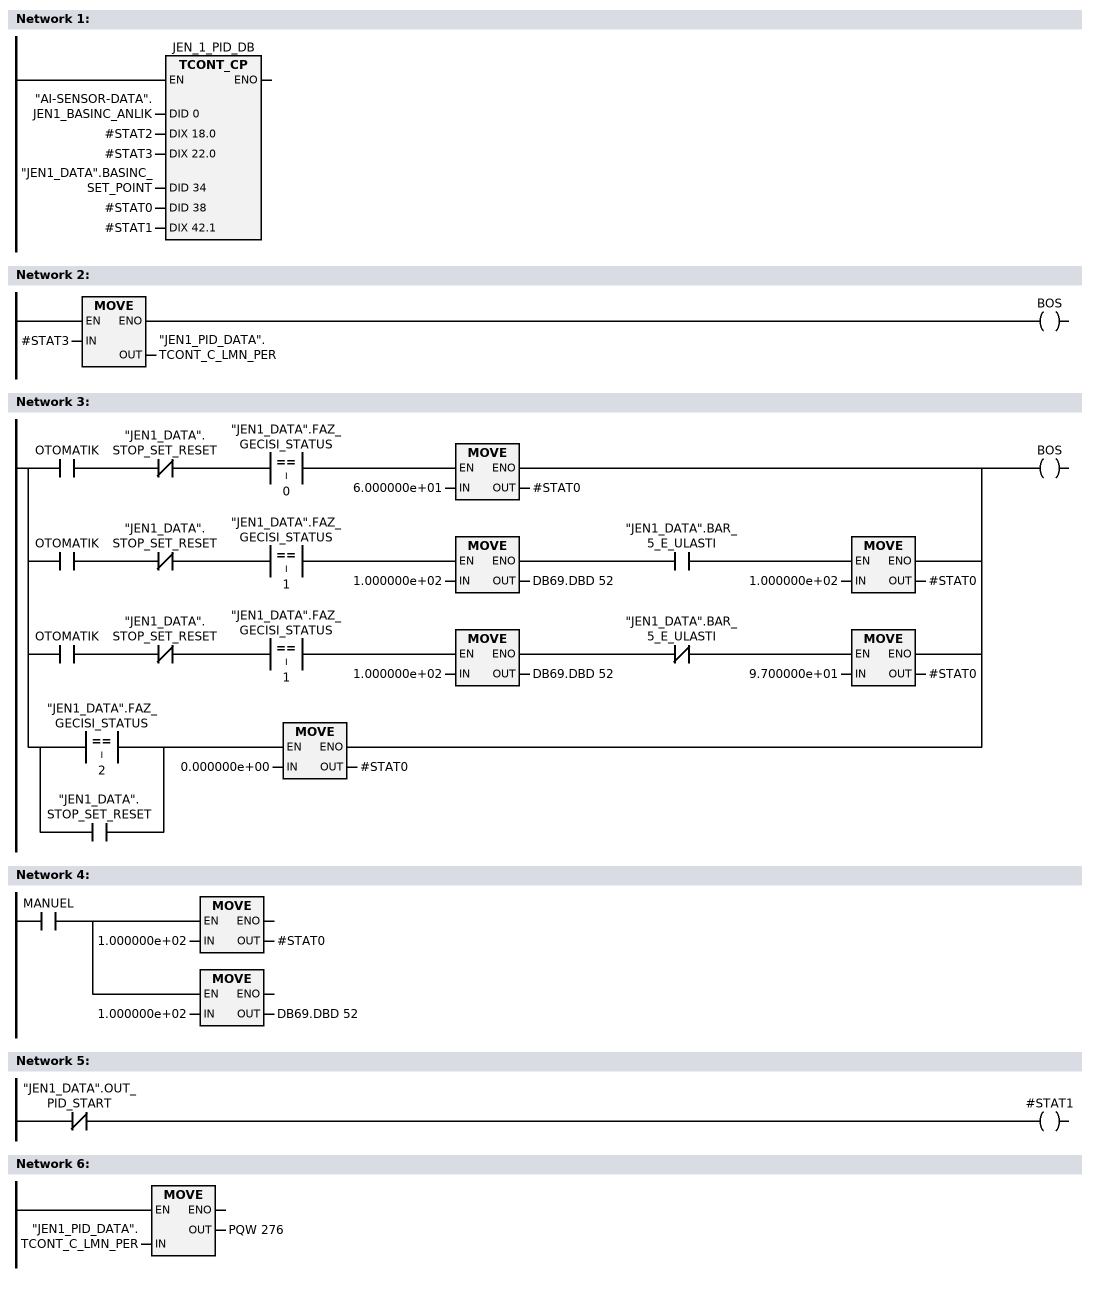
NETWORK
TITLE =
      CALL  "TCONT_CP" , "JEN_1_PID_DB" (
           DID 0                    := "AI-SENSOR-DATA".JEN1_BASINC_ANLIK,
           DIX 18.0                 := #STAT2,
           DIX 22.0                 := #STAT3,
           DID 34                   := "JEN1_DATA".BASINC_SET_POINT,
           DID 38                   := #STAT0,
           DIX 42.1                 := #STAT1);
      NOP   0;
NETWORK
TITLE =
      L     #STAT3;
      T     "JEN1_PID_DATA".TCONT_C_LMN_PER;
      SET;
      SAVE;
      CLR;
      A     BR;
      =     "BOS";
NETWORK
TITLE =
      O(;
      A     "OTOMATIK";
      AN    "JEN1_DATA".STOP_SET_RESET;
      A(;
      L     "JEN1_DATA".FAZ_GECISI_STATUS;
      L     0;
      ==I;
      );
      JNB   _001;
      L     6.000000e+01;
      T     #STAT0;
      SET;
      SAVE;
      CLR;
_001: A     BR;
      );
      O(;
      A(;
      A     "OTOMATIK";
      AN    "JEN1_DATA".STOP_SET_RESET;
      A(;
      L     "JEN1_DATA".FAZ_GECISI_STATUS;
      L     1;
      ==I;
      );
      JNB   _002;
      L     1.000000e+02;
      T     DB69.DBD 52;
      SET;
      SAVE;
      CLR;
_002: A     BR;
      );
      A     "JEN1_DATA".BAR_5_E_ULASTI;
      JNB   _003;
      L     1.000000e+02;
      T     #STAT0;
      SET;
      SAVE;
      CLR;
_003: A     BR;
      );
      O(;
      A(;
      A     "OTOMATIK";
      AN    "JEN1_DATA".STOP_SET_RESET;
      A(;
      L     "JEN1_DATA".FAZ_GECISI_STATUS;
      L     1;
      ==I;
      );
      JNB   _004;
      L     1.000000e+02;
      T     DB69.DBD 52;
      SET;
      SAVE;
      CLR;
_004: A     BR;
      );
      AN    "JEN1_DATA".BAR_5_E_ULASTI;
      JNB   _005;
      L     9.700000e+01;
      T     #STAT0;
      SET;
      SAVE;
      CLR;
_005: A     BR;
      );
      O(;
      A(;
      O(;
      L     "JEN1_DATA".FAZ_GECISI_STATUS;
      L     2;
      ==I;
      );
      O     "JEN1_DATA".STOP_SET_RESET;
      );
      JNB   _006;
      L     0.000000e+00;
      T     #STAT0;
      SET;
      SAVE;
      CLR;
_006: A     BR;
      );
      =     "BOS";
NETWORK
TITLE =
      A     "MANUEL";
      =     L 0.0;
      A     L 0.0;
      JNB   _007;
      L     1.000000e+02;
      T     #STAT0;
_007: NOP   0;
      A     L 0.0;
      JNB   _008;
      L     1.000000e+02;
      T     DB69.DBD 52;
_008: NOP   0;
NETWORK
TITLE =
      AN    "JEN1_DATA".OUT_PID_START;
      =     #STAT1;
NETWORK
TITLE =
      L     "JEN1_PID_DATA".TCONT_C_LMN_PER;
      T     PQW 276;
      NOP   0;
END_FUNCTION_BLOCK

FUNCTION_BLOCK "JEN2_PID_KONTROL"	// FB 50
VERSION : 0.1
VAR
  STAT0 : REAL ;
  STAT1 : INT ;
  STAT2 : REAL ;
  STAT3 : BOOL ;
  STAT4 : BOOL ;
END_VAR
BEGIN
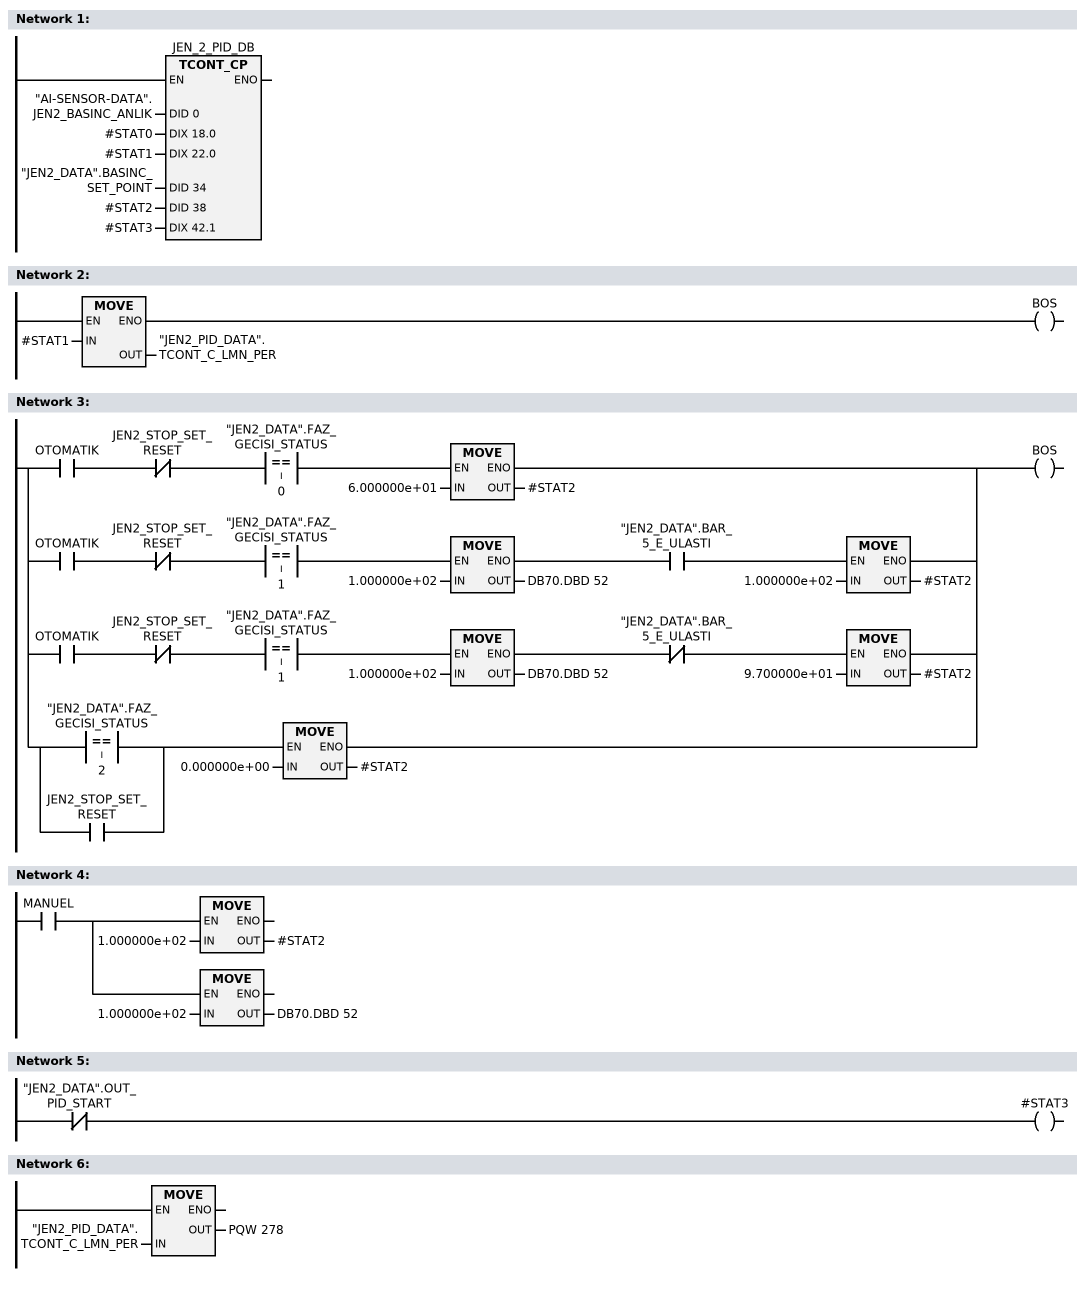
NETWORK
TITLE =
      CALL  "TCONT_CP" , "JEN_2_PID_DB" (
           DID 0                    := "AI-SENSOR-DATA".JEN2_BASINC_ANLIK,
           DIX 18.0                 := #STAT0,
           DIX 22.0                 := #STAT1,
           DID 34                   := "JEN2_DATA".BASINC_SET_POINT,
           DID 38                   := #STAT2,
           DIX 42.1                 := #STAT3);
      NOP   0;
NETWORK
TITLE =
      L     #STAT1;
      T     "JEN2_PID_DATA".TCONT_C_LMN_PER;
      SET;
      SAVE;
      CLR;
      A     BR;
      =     "BOS";
NETWORK
TITLE =
      O(;
      A     "OTOMATIK";
      AN    "JEN2_STOP_SET_RESET";
      A(;
      L     "JEN2_DATA".FAZ_GECISI_STATUS;
      L     0;
      ==I;
      );
      JNB   _001;
      L     6.000000e+01;
      T     #STAT2;
      SET;
      SAVE;
      CLR;
_001: A     BR;
      );
      O(;
      A(;
      A     "OTOMATIK";
      AN    "JEN2_STOP_SET_RESET";
      A(;
      L     "JEN2_DATA".FAZ_GECISI_STATUS;
      L     1;
      ==I;
      );
      JNB   _002;
      L     1.000000e+02;
      T     DB70.DBD 52;
      SET;
      SAVE;
      CLR;
_002: A     BR;
      );
      A     "JEN2_DATA".BAR_5_E_ULASTI;
      JNB   _003;
      L     1.000000e+02;
      T     #STAT2;
      SET;
      SAVE;
      CLR;
_003: A     BR;
      );
      O(;
      A(;
      A     "OTOMATIK";
      AN    "JEN2_STOP_SET_RESET";
      A(;
      L     "JEN2_DATA".FAZ_GECISI_STATUS;
      L     1;
      ==I;
      );
      JNB   _004;
      L     1.000000e+02;
      T     DB70.DBD 52;
      SET;
      SAVE;
      CLR;
_004: A     BR;
      );
      AN    "JEN2_DATA".BAR_5_E_ULASTI;
      JNB   _005;
      L     9.700000e+01;
      T     #STAT2;
      SET;
      SAVE;
      CLR;
_005: A     BR;
      );
      O(;
      A(;
      O(;
      L     "JEN2_DATA".FAZ_GECISI_STATUS;
      L     2;
      ==I;
      );
      O     "JEN2_STOP_SET_RESET";
      );
      JNB   _006;
      L     0.000000e+00;
      T     #STAT2;
      SET;
      SAVE;
      CLR;
_006: A     BR;
      );
      =     "BOS";
NETWORK
TITLE =
      A     "MANUEL";
      =     L 0.0;
      A     L 0.0;
      JNB   _007;
      L     1.000000e+02;
      T     #STAT2;
_007: NOP   0;
      A     L 0.0;
      JNB   _008;
      L     1.000000e+02;
      T     DB70.DBD 52;
_008: NOP   0;
NETWORK
TITLE =
      AN    "JEN2_DATA".OUT_PID_START;
      =     #STAT3;
NETWORK
TITLE =
      L     "JEN2_PID_DATA".TCONT_C_LMN_PER;
      T     PQW 278;
      NOP   0;
END_FUNCTION_BLOCK

// FB 58: know-how protected block, not included

FUNCTION_BLOCK "KAZAN_1_KONTROL"	// FB 94
VERSION : 0.1
BEGIN
NETWORK
TITLE =
      CALL  "Int_To_S5Time" (
           Saat                     := "HMI_DATA".Otoklav_1_TimeData.Hours,
           Dakika                   := "HMI_DATA".Otoklav_1_TimeData.Minutes,
           HesaplananSure_S5TIME    := "KAZAN1_DATA".IN_PISIM_SURESI);
      CALL  "KAZAN_ORTAK" , DB 120 (
           IN_ACIL_STOP             := "KAZAN1_ACIL_STOP",
           IN_START                 := "KAZAN1_START",
           IN_TRANSFER              := "KAZAN1_TRANSFER",
           IN_BOSALTIM              := "KAZAN1_BOSALTIM",
           IN_KAPAK                 := "KAZAN1_KAPAK_SW",
           IN_JENS_OK               := "KAZAN1_DATA".IN_JEN_OK,
           IN_TRANSFERE_HAZIR       := "KAZAN1_DATA".IN_DIGER_KAZ_TRANS_HAZIR,
           IN_PISIM_SURESI          := "KAZAN1_DATA".IN_PISIM_SURESI,
           IN_SCALE_BASINC_PER      := "KAZAN1_DATA".IN_SCALE_BASINC_PER,
           IN_SET_BASINC            := "KAZAN1_DATA".IN_SET_BASINC,
           IN_DIGER_KAZAN_BASINCI   := "KAZAN1_DATA".IN_DIGER_KAZAN_BASINCI,
           IN_TIMER_500MS           := "500ms_delay1",
           IN_TIMER_1S              := "1s Delay",
           IN_TIMER_PISIRME         := "Pisim_Suresi",
           IN_TIMER_500MS_2         := "500ms_delay",
           IN_TIMER_7S              := "s_offt_7s_delay",
           IN_SCALE_HI_LIM          := 1.000000e+01,
           IN_SCALE_LO_LIM          := 0.000000e+00,
           IN_SCALE_SICAKLIK_HI_LIM := 2.000000e+02,
           IN_SCALE_SICAKLIK_LO_LIM := 0.000000e+00,
           IN_SCALE_SICAKLIK_PER    := "KAZAN1_DATA".IN_SCALE_SICAKLIK_PER,
           IN_DIGER_KAZAN_BOSALTIMD := "KAZAN1_DATA".IN_DIGER_KAZ_BOSALTIMDA,
           IN_TRANSFER_BASLADI      := "KAZAN1_DATA".IN_DIGER_KAZ_TRANSFERDE,
           IN_JEN_DURDU             := "ORTAK_DATA".OTO_ISLEM_BITTI_VANA_AC,
           IN_DELAY_BITISI_BEKLE    := "OTO_1_DELAY_PISIM_BITTI",
           IN_DELAY_BIRAZ_BEKLE     := "DELAY_ADIM5_BEKLE",
           IN31                     := T 58,
           IN32                     := T 61,
           Bos_Vana_Period_Timer    := T 3,
           Bos_Vana_Aciklik_Timer   := T 4,
           BosVana_Per_TimeInterval := "HMI_DATA".Otoklav1_Bos_Vanasi.Periyod_Bekleme_Suresi,
           BosVana_Aci_TimeInterval := "HMI_DATA".Otoklav1_Bos_Vanasi.Acik_Kalma_Suresi,
           BosVana_Acik_Sayisi      := "HMI_DATA".Otoklav1_Bos_Vanasi.Vana_Acilma_Sayisi,
           O_YESIL_LAM              := "KAZAN1_YESIL_LAMBA",
           O_KIRMIZI_LAM            := "KAZAN1_KIRMIZI_LAMBA",
           O_DUDUK                  := "KAZAN1_DUDUK",
           O_BOSALTIM_VALFI         := "KAZAN1_BOSALTIM_VALFI",
           O_PID_MAN_ON             := "KAZAN1_DATA".O_PID_MAN_ON,
           O_PID_MAN                := "KAZAN1_DATA".O_PID_MAN,
           O_TRANSFER_YAPILIYOR     := "KAZAN1_DATA".O_TRANSFER_YAPILIYOR,
           O_SCALE_BASINC_RET_VAL   := "KAZAN1_DATA".O_SCALE_BASINC_RET_VAL,
           O_SCALE_BASINC_OUT       := "KAZAN1_DATA".O_SCALE_BASINC_OUT,
           O_EMNIYET_VALFI          := "KAZAN1_EMN_VALFI_BOS",
           O_TRANSFERE_HAZIR        := "KAZAN1_DATA".O_TRANSFERE_HAZIR,
           O_SCALE_SICAKLIK_RET_VAL := "KAZAN1_DATA".O_SCALE_SICAKLIK_RET_VAL,
           O_SCALE_SICAKLIK_OUT     := "KAZAN1_DATA".O_SCALE_SICAKLIK_OUT,
           O_TRANSFER_ET_LAMBASI    := "KAZAN1_TRANS_BUT_LAMBASI",
           O_PROSES_BASLADI         := M 300.0,
           O_KAZAN_BOSALTIMDA       := "KAZAN1_DATA".O_KAZAN_BOSALTIMDA,
           O_PISIM_BASLADI          := "KAZAN1_DATA".O_PISIM_BASLADI,
           STATUS                   := "KAZAN1_DATA".IN_STATUS);
//       IN0  :="KAZAN1_ACIL_STOP"
//       IN1  :="KAZAN1_START"
//       IN2  :="KAZAN1_TRANSFER"
//       IN3  :="KAZAN1_BOSALTIM"
//       IN4  :="KAZAN1_KAPAK_SW"
//       IN5  :=
//       IN6  :=
//       IN7  :="KAZAN1_DATA".IN_JEN_OK
//       IN8  :="KAZAN1_DATA".IN_DIGER_KAZ_TRANS_HAZIR
//       IN9  :="KAZAN1_DATA".IN_PISIM_SURESI
//       IN10 :="KAZAN1_DATA".IN_SCALE_BASINC_PER
//       IN11 :="KAZAN1_DATA".IN_SET_BASINC
//       IN12 :="KAZAN1_DATA".IN_DIGER_KAZAN_BASINCI
//       IN13 :="500ms_delay1"
//       IN14 :="1s Delay"
//       IN15 :="Pisim_Suresi"
//       IN16 :="500ms_delay"
//       IN17 :="s_offt_7s_delay"
//       IN18 :=1.000000e+001
//       IN19 :=0.000000e+000
//       IN20 :=2.000000e+002
//       IN21 :=0.000000e+000
//       IN22 :="KAZAN1_DATA".IN_SCALE_SICAKLIK_PER
//       IN23 :="KAZAN1_DATA".IN_DIGER_KAZ_BOSALTIMDA
//       IN24 :="KAZAN1_DATA".IN_DIGER_KAZ_TRANSFERDE
//       IN25 :=
//       IN26 :=
//       IN27 :="ORTAK_DATA".OTO_ISLEM_BITTI_VANA_AC
//       IN28 :=
//       IN29 :="OTO_1_DELAY_PISIM_BITTI"
//       IN30 :="DELAY_ADIM5_BEKLE"
//       IN31 :=T58
//       IN32 :=T61
//       OUT33:="KAZAN1_YESIL_LAMBA"
//       OUT34:="KAZAN1_KIRMIZI_LAMBA"
//       OUT35:="KAZAN1_DUDUK"
//       OUT36:="KAZAN1_BOSALTIM_VALFI"
//       OUT37:="KAZAN1_DATA".O_PID_MAN_ON
//       OUT38:="KAZAN1_DATA".O_PID_MAN
//       OUT39:="KAZAN1_DATA".O_TRANSFER_YAPILIYOR
//       OUT40:="KAZAN1_DATA".O_SCALE_BASINC_RET_VAL
//       OUT41:="KAZAN1_DATA".O_SCALE_BASINC_OUT
//       OUT42:="KAZAN1_EMN_VALFI_BOS"
//       OUT43:="KAZAN1_DATA".O_TRANSFERE_HAZIR
//       OUT44:="KAZAN1_DATA".O_SCALE_SICAKLIK_RET_VAL
//       OUT45:="KAZAN1_DATA".O_SCALE_SICAKLIK_OUT
//       OUT46:="KAZAN1_TRANS_BUT_LAMBASI"
//       OUT47:=M300.0
//       OUT48:="KAZAN1_DATA".O_KAZAN_BOSALTIMDA
//       OUT49:="KAZAN1_DATA".O_PISIM_BASLADI
//       IO50 :="KAZAN1_DATA".IN_STATUS
NETWORK
TITLE =
      A     "KAZAN2_DATA".O_TRANSFERE_HAZIR;
      =     "KAZAN1_DATA".IN_DIGER_KAZ_TRANS_HAZIR;
      L     PIW 272;
      T     "KAZAN1_DATA".IN_SCALE_BASINC_PER;
      L     PIW 274;
      T     "KAZAN1_DATA".IN_SCALE_SICAKLIK_PER;
      L     "KAZAN2_DATA".O_SCALE_BASINC_OUT;
      T     "KAZAN1_DATA".IN_DIGER_KAZAN_BASINCI;
      O     "JEN1_DATA".JEN1_HAZIR;
      O     "JEN2_DATA".JEN2_HAZIR;
      =     "KAZAN1_DATA".IN_JEN_OK;
      A     "KAZAN2_DATA".O_KAZAN_BOSALTIMDA;
      =     "KAZAN1_DATA".IN_DIGER_KAZ_BOSALTIMDA;
      A     "KAZAN2_DATA".O_TRANSFER_YAPILIYOR;
      =     "KAZAN1_DATA".IN_DIGER_KAZ_TRANSFERDE;
END_FUNCTION_BLOCK

FUNCTION_BLOCK "KAZAN_2_KONTROL"	// FB 95
VERSION : 0.1
BEGIN
NETWORK
TITLE =
      CALL  "Int_To_S5Time" (
           Saat                     := "HMI_DATA".Otoklav_2_TimeData.Hours,
           Dakika                   := "HMI_DATA".Otoklav_2_TimeData.Minutes,
           HesaplananSure_S5TIME    := "KAZAN2_DATA".IN_PISIM_SURESI);
      CALL  "KAZAN_ORTAK" , DB 230 (
           IN_ACIL_STOP             := "KAZAN2_ACIL_STOP",
           IN_START                 := "KAZAN2_START",
           IN_TRANSFER              := "KAZAN2_TRANSFER",
           IN_BOSALTIM              := "KAZAN2_BOSALTIM",
           IN_KAPAK                 := "KAZAN2_KAPAK_SW",
           IN_JENS_OK               := "KAZAN2_DATA".IN_JEN_OK,
           IN_TRANSFERE_HAZIR       := "KAZAN2_DATA".IN_DIGER_KAZ_TRANS_HAZIR,
           IN_PISIM_SURESI          := "KAZAN2_DATA".IN_PISIM_SURESI,
           IN_SCALE_BASINC_PER      := "KAZAN2_DATA".IN_SCALE_BASINC_PER,
           IN_SET_BASINC            := "KAZAN2_DATA".IN_SET_BASINC,
           IN_DIGER_KAZAN_BASINCI   := "KAZAN2_DATA".IN_DIGER_KAZAN_BASINCI,
           IN_TIMER_500MS           := "500ms_delay_kazan_2",
           IN_TIMER_1S              := "1ms_delay_kazan_2",
           IN_TIMER_PISIRME         := "kazan_2_pisirme_delay",
           IN_TIMER_500MS_2         := "kazan_2_500ms_delay",
           IN_TIMER_7S              := "kazan_2_7s_delay",
           IN_SCALE_HI_LIM          := 1.000000e+01,
           IN_SCALE_LO_LIM          := 0.000000e+00,
           IN_SCALE_SICAKLIK_HI_LIM := 2.000000e+02,
           IN_SCALE_SICAKLIK_LO_LIM := 0.000000e+00,
           IN_SCALE_SICAKLIK_PER    := "KAZAN2_DATA".IN_SCALE_SICAKLIK_PER,
           IN_DIGER_KAZAN_BOSALTIMD := "KAZAN2_DATA".IN_DIGER_KAZ_BOSALTIMDA,
           IN_TRANSFER_BASLADI      := "KAZAN2_DATA".IN_DIGER_KAZ_TRANSFERDE,
           IN_JEN_DURDU             := "ORTAK_DATA".OTO_ISLEM_BITTI_VANA_AC,
           IN_DELAY_BITISI_BEKLE    := "OTO_2_DELAY_BITIS",
           IN_DELAY_BIRAZ_BEKLE     := "DELAY_ADIM5_BEKLE2",
           IN31                     := T 60,
           IN32                     := T 62,
           Bos_Vana_Period_Timer    := T 5,
           Bos_Vana_Aciklik_Timer   := T 7,
           BosVana_Per_TimeInterval := "HMI_DATA".Otoklav2_Bos_Vanasi.Periyod_Bekleme_Suresi,
           BosVana_Aci_TimeInterval := "HMI_DATA".Otoklav2_Bos_Vanasi.Acik_Kalma_Suresi,
           BosVana_Acik_Sayisi      := "HMI_DATA".Otoklav2_Bos_Vanasi.Vana_Acilma_Sayisi,
           O_YESIL_LAM              := "KAZAN2_YESIL_LAMBA",
           O_KIRMIZI_LAM            := "KAZAN2_KIRMIZI_LAMBA",
           O_DUDUK                  := "KAZAN2_DUDUK",
           O_BOSALTIM_VALFI         := "KAZAN2_BOSALTIM_VALFI",
           O_PID_MAN_ON             := "KAZAN2_DATA".O_PID_MAN_ON,
           O_PID_MAN                := "KAZAN2_DATA".O_PID_MAN,
           O_TRANSFER_YAPILIYOR     := "KAZAN2_DATA".O_TRANSFER_YAPILIYOR,
           O_SCALE_BASINC_RET_VAL   := "KAZAN2_DATA".O_SCALE_BASINC_RET_VAL,
           O_SCALE_BASINC_OUT       := "KAZAN2_DATA".O_SCALE_BASINC_OUT,
           O_EMNIYET_VALFI          := "KAZAN2_EMN_VALFI_BOS",
           O_TRANSFERE_HAZIR        := "KAZAN2_DATA".O_TRANSFERE_HAZIR,
           O_SCALE_SICAKLIK_RET_VAL := "KAZAN2_DATA".O_SCALE_SICAKLIK_RET_VAL,
           O_SCALE_SICAKLIK_OUT     := "KAZAN2_DATA".O_SCALE_SICAKLIK_OUT,
           O_TRANSFER_ET_LAMBASI    := "KAZAN2_TRANS_BUT_LAMBASI",
           O_PROSES_BASLADI         := M 300.1,
           O_KAZAN_BOSALTIMDA       := "KAZAN2_DATA".O_KAZAN_BOSALTIMDA,
           O_PISIM_BASLADI          := "KAZAN2_DATA".O_PISIM_BASLADI,
           STATUS                   := "KAZAN2_DATA".IN_STATUS);
//      CALL  "KAZAN_ORTAK" , DB230
//       IN0  :="KAZAN2_ACIL_STOP"
//       IN1  :="KAZAN2_START"
//       IN2  :="KAZAN2_TRANSFER"
//       IN3  :="KAZAN2_BOSALTIM"
//       IN4  :="KAZAN2_KAPAK_SW"
//       IN5  :=
//       IN6  :=
//       IN7  :="KAZAN2_DATA".IN_JEN_OK
//       IN8  :="KAZAN2_DATA".IN_DIGER_KAZ_TRANS_HAZIR
//       IN9  :="KAZAN2_DATA".IN_PISIM_SURESI
//       IN10 :="KAZAN2_DATA".IN_SCALE_BASINC_PER
//       IN11 :="KAZAN2_DATA".IN_SET_BASINC
//       IN12 :="KAZAN2_DATA".IN_DIGER_KAZAN_BASINCI
//       IN13 :="500ms_delay_kazan_2"
//       IN14 :="1ms_delay_kazan_2"
//       IN15 :="kazan_2_pisirme_delay"
//       IN16 :="kazan_2_500ms_delay"
//       IN17 :="kazan_2_7s_delay"
//       IN18 :=1.000000e+001
//       IN19 :=0.000000e+000
//       IN20 :=2.000000e+002
//       IN21 :=0.000000e+000
//       IN22 :="KAZAN2_DATA".IN_SCALE_SICAKLIK_PER
//       IN23 :="KAZAN2_DATA".IN_DIGER_KAZ_BOSALTIMDA
//       IN24 :="KAZAN2_DATA".IN_DIGER_KAZ_TRANSFERDE
//       IN25 :=
//       IN26 :=
//       IN27 :="ORTAK_DATA".OTO_ISLEM_BITTI_VANA_AC
//       IN28 :=
//       IN29 :="OTO_2_DELAY_BITIS"
//       IN30 :="DELAY_ADIM5_BEKLE2"
//       IN31 :=T60
//       IN32 :=T62
//       OUT33:="KAZAN2_YESIL_LAMBA"
//       OUT34:="KAZAN2_KIRMIZI_LAMBA"
//       OUT35:="KAZAN2_DUDUK"
//       OUT36:="KAZAN2_BOSALTIM_VALFI"
//       OUT37:="KAZAN2_DATA".O_PID_MAN_ON
//       OUT38:="KAZAN2_DATA".O_PID_MAN
//       OUT39:="KAZAN2_DATA".O_TRANSFER_YAPILIYOR
//       OUT40:="KAZAN2_DATA".O_SCALE_BASINC_RET_VAL
//       OUT41:="KAZAN2_DATA".O_SCALE_BASINC_OUT
//       OUT42:="KAZAN2_EMN_VALFI_BOS"
//       OUT43:="KAZAN2_DATA".O_TRANSFERE_HAZIR
//       OUT44:="KAZAN2_DATA".O_SCALE_SICAKLIK_RET_VAL
//       OUT45:="KAZAN2_DATA".O_SCALE_SICAKLIK_OUT
//       OUT46:="KAZAN2_TRANS_BUT_LAMBASI"
//       OUT47:=M300.1
//       OUT48:="KAZAN2_DATA".O_KAZAN_BOSALTIMDA
//       OUT49:="KAZAN2_DATA".O_PISIM_BASLADI
//       IO50 :="KAZAN2_DATA".IN_STATUS
NETWORK
TITLE =
      A     "KAZAN1_DATA".O_TRANSFERE_HAZIR;
      =     "KAZAN2_DATA".IN_DIGER_KAZ_TRANS_HAZIR;
      L     PIW 276;
      T     "KAZAN2_DATA".IN_SCALE_BASINC_PER;
      L     PIW 278;
      T     "KAZAN2_DATA".IN_SCALE_SICAKLIK_PER;
      L     "KAZAN1_DATA".O_SCALE_BASINC_OUT;
      T     "KAZAN2_DATA".IN_DIGER_KAZAN_BASINCI;
      O     "JEN1_DATA".JEN1_HAZIR;
      O     "JEN2_DATA".JEN2_HAZIR;
      =     "KAZAN2_DATA".IN_JEN_OK;
      A     "KAZAN1_DATA".O_KAZAN_BOSALTIMDA;
      =     "KAZAN2_DATA".IN_DIGER_KAZ_BOSALTIMDA;
      A     "KAZAN1_DATA".O_TRANSFER_YAPILIYOR;
      =     "KAZAN2_DATA".IN_DIGER_KAZ_TRANSFERDE;
END_FUNCTION_BLOCK

FUNCTION_BLOCK "JEN1_KONTROL_BLOGU"	// FB 98
VERSION : 0.1
VAR
  STAT0 : BOOL ;
  STAT1 : BOOL ;
  STAT2 : BOOL ;
  STAT3 : BOOL ;
  STAT4 : BOOL ;
END_VAR
VAR_TEMP
  TEMP5 : BOOL ;
  TEMP6 : BOOL ;
  TEMP7 : BOOL ;
  TEMP8 : BOOL ;
  TEMP9 : BOOL ;
  TEMP10 : BOOL ;
  TEMP11 : BOOL ;
  TEMP12 : BOOL ;
  TEMP13 : BOOL ;
  TEMP14 : BOOL ;
  TEMP15 : BOOL ;
  TEMP16 : BOOL ;
END_VAR
BEGIN
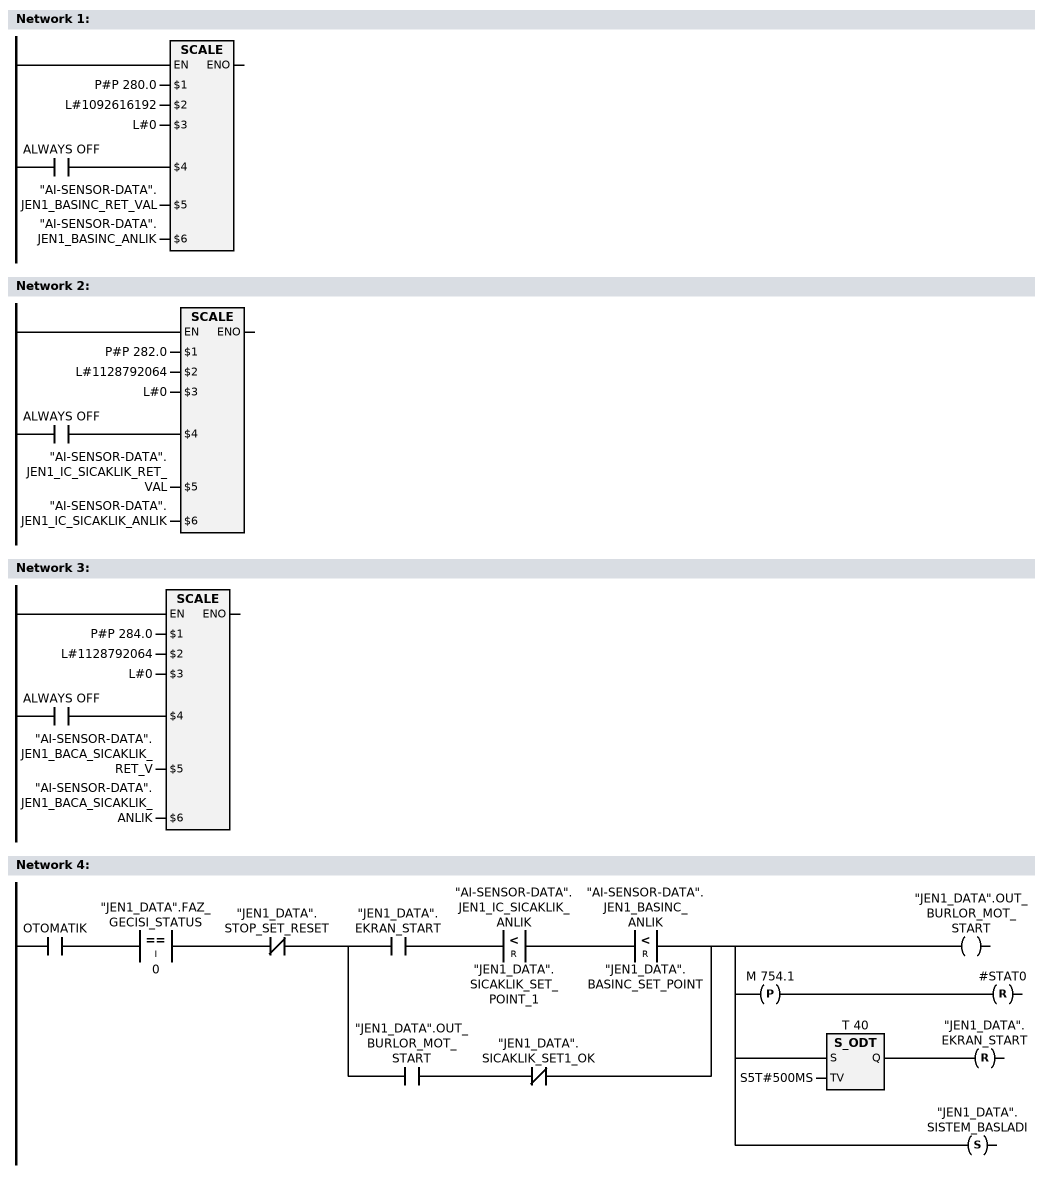
NETWORK
TITLE =
      A     "ALWAYS OFF";
      =     L 2.0;
      BLD   103;
      CALL  "SCALE" (
           $1                       := P#P 280.0,
           $2                       := L#1092616192,
           $3                       := L#0,
           $4                       := L 2.0,
           $5                       := "AI-SENSOR-DATA".JEN1_BASINC_RET_VAL,
           $6                       := "AI-SENSOR-DATA".JEN1_BASINC_ANLIK);
      NOP   0;
NETWORK
TITLE =
      A     "ALWAYS OFF";
      =     L 2.0;
      BLD   103;
      CALL  "SCALE" (
           $1                       := P#P 282.0,
           $2                       := L#1128792064,
           $3                       := L#0,
           $4                       := L 2.0,
           $5                       := "AI-SENSOR-DATA".JEN1_IC_SICAKLIK_RET_VAL,
           $6                       := "AI-SENSOR-DATA".JEN1_IC_SICAKLIK_ANLIK);
      NOP   0;
NETWORK
TITLE =
      A     "ALWAYS OFF";
      =     L 2.0;
      BLD   103;
      CALL  "SCALE" (
           $1                       := P#P 284.0,
           $2                       := L#1128792064,
           $3                       := L#0,
           $4                       := L 2.0,
           $5                       := "AI-SENSOR-DATA".JEN1_BACA_SICAKLIK_RET_V,
           $6                       := "AI-SENSOR-DATA".JEN1_BACA_SICAKLIK_ANLIK);
      NOP   0;
NETWORK
TITLE =
      A     "OTOMATIK";
      A(;
      L     "JEN1_DATA".FAZ_GECISI_STATUS;
      L     0;
      ==I;
      );
      AN    "JEN1_DATA".STOP_SET_RESET;
      A(;
      A     "JEN1_DATA".EKRAN_START;
      A(;
      L     "AI-SENSOR-DATA".JEN1_IC_SICAKLIK_ANLIK;
      L     "JEN1_DATA".SICAKLIK_SET_POINT_1;
      <R;
      );
      A(;
      L     "AI-SENSOR-DATA".JEN1_BASINC_ANLIK;
      L     "JEN1_DATA".BASINC_SET_POINT;
      <R;
      );
      O;
      A     "JEN1_DATA".OUT_BURLOR_MOT_START;
      AN    "JEN1_DATA".SICAKLIK_SET1_OK;
      );
      =     L 2.0;
      A     L 2.0;
      BLD   102;
      =     "JEN1_DATA".OUT_BURLOR_MOT_START;
      A     L 2.0;
      FP    M 754.1;
      R     #STAT0;
      A     L 2.0;
      L     S5T#500MS;
      SD    T 40;
      NOP   0;
      NOP   0;
      NOP   0;
      A     T 40;
      R     "JEN1_DATA".EKRAN_START;
      A     L 2.0;
      BLD   102;
      S     "JEN1_DATA".SISTEM_BASLADI;
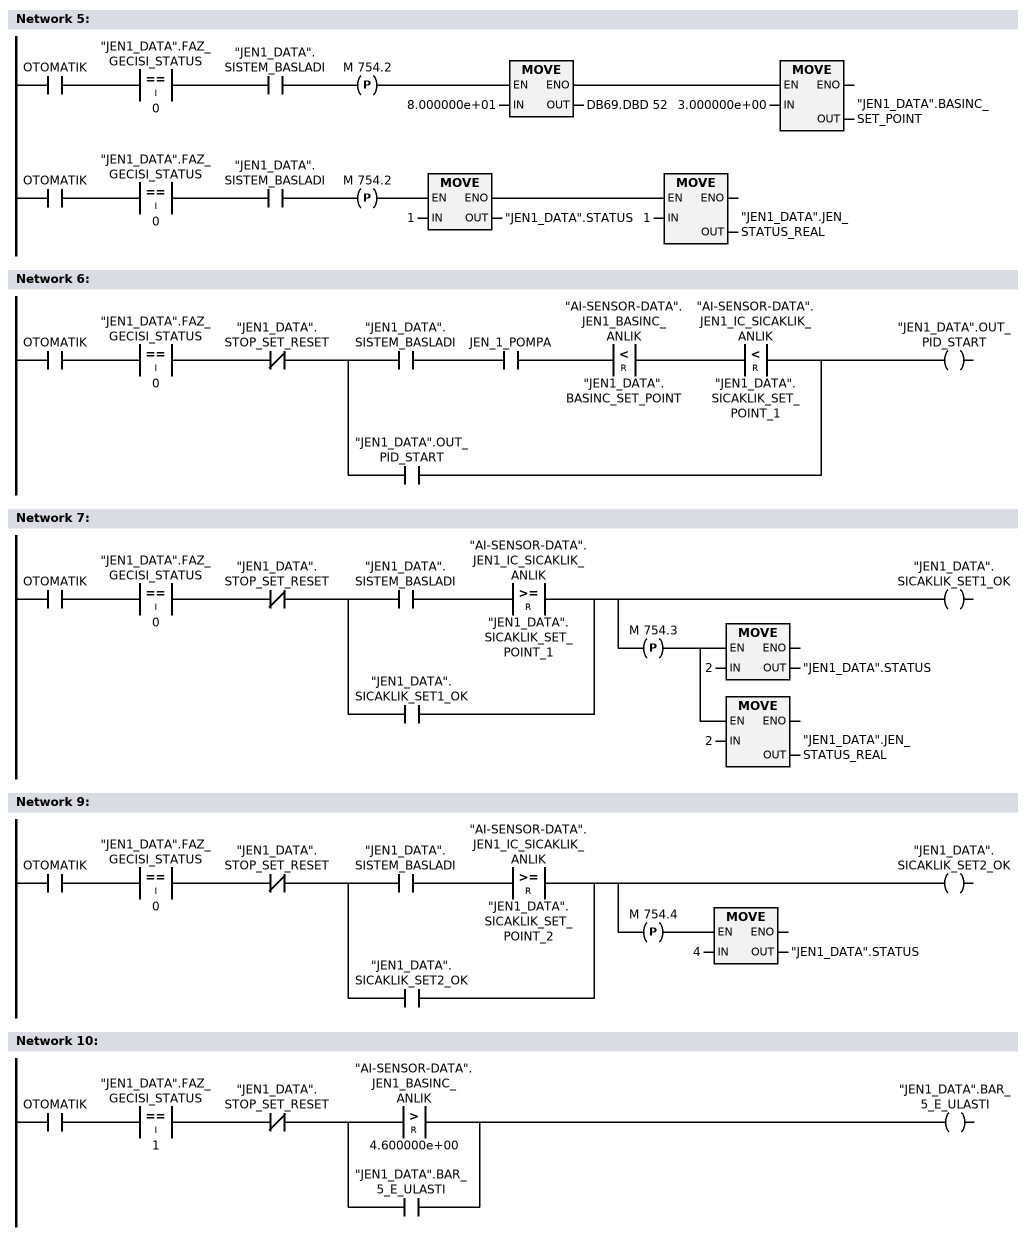
NETWORK
TITLE =
      A     "OTOMATIK";
      A(;
      L     "JEN1_DATA".FAZ_GECISI_STATUS;
      L     0;
      ==I;
      );
      A     "JEN1_DATA".SISTEM_BASLADI;
      FP    M 754.2;
      =     L 2.0;
      A(;
      A     L 2.0;
      JNB   _001;
      L     8.000000e+01;
      T     DB69.DBD 52;
      SET;
      SAVE;
      CLR;
_001: A     BR;
      );
      JNB   _002;
      L     3.000000e+00;
      T     "JEN1_DATA".BASINC_SET_POINT;
_002: NOP   0;
      A(;
      A     L 2.0;
      JNB   _003;
      L     1;
      T     "JEN1_DATA".STATUS;
      SET;
      SAVE;
      CLR;
_003: A     BR;
      );
      JNB   _004;
      L     1;
      T     "JEN1_DATA".JEN_STATUS_REAL;
_004: NOP   0;
NETWORK
TITLE =
      A     "OTOMATIK";
      A(;
      L     "JEN1_DATA".FAZ_GECISI_STATUS;
      L     0;
      ==I;
      );
      AN    "JEN1_DATA".STOP_SET_RESET;
      A(;
      A     "JEN1_DATA".SISTEM_BASLADI;
      A     "JEN_1_POMPA";
      A(;
      L     "AI-SENSOR-DATA".JEN1_BASINC_ANLIK;
      L     "JEN1_DATA".BASINC_SET_POINT;
      <R;
      );
      A(;
      L     "AI-SENSOR-DATA".JEN1_IC_SICAKLIK_ANLIK;
      L     "JEN1_DATA".SICAKLIK_SET_POINT_1;
      <R;
      );
      O     "JEN1_DATA".OUT_PID_START;
      );
      =     "JEN1_DATA".OUT_PID_START;
NETWORK
TITLE =
      A     "OTOMATIK";
      A(;
      L     "JEN1_DATA".FAZ_GECISI_STATUS;
      L     0;
      ==I;
      );
      AN    "JEN1_DATA".STOP_SET_RESET;
      A(;
      A     "JEN1_DATA".SISTEM_BASLADI;
      A(;
      L     "AI-SENSOR-DATA".JEN1_IC_SICAKLIK_ANLIK;
      L     "JEN1_DATA".SICAKLIK_SET_POINT_1;
      >=R;
      );
      O     "JEN1_DATA".SICAKLIK_SET1_OK;
      );
      =     L 2.0;
      A     L 2.0;
      BLD   102;
      =     "JEN1_DATA".SICAKLIK_SET1_OK;
      A     L 2.0;
      FP    M 754.3;
      =     L 2.1;
      A     L 2.1;
      JNB   _005;
      L     2;
      T     "JEN1_DATA".STATUS;
_005: NOP   0;
      A     L 2.1;
      JNB   _006;
      L     2;
      T     "JEN1_DATA".JEN_STATUS_REAL;
_006: NOP   0;
NETWORK
TITLE =
      A(;
      A     "JEN1_DATA".SICAKLIK_SET1_OK;
      FP    "SET2_ULASMADI_RIS";
      S     "SET2_ULASMADI_SR";
      A(;
      O(;
      L     "JEN1_DATA".FAZ_GECISI_STATUS;
      L     1;
      ==I;
      );
      O     "JEN1_DATA".STOP_SET_RESET;
      );
      R     "SET2_ULASMADI_SR";
      A     "SET2_ULASMADI_SR";
      );
      L     S5T#1M30S;
      SD    "TIM_SET2_ULASMADI";
      NOP   0;
      NOP   0;
      NOP   0;
      A     "TIM_SET2_ULASMADI";
      =     "JEN1_DATA".SET2_DEGERINE_ULASMADI;
NETWORK
TITLE =
      A     "OTOMATIK";
      A(;
      L     "JEN1_DATA".FAZ_GECISI_STATUS;
      L     0;
      ==I;
      );
      AN    "JEN1_DATA".STOP_SET_RESET;
      A(;
      A     "JEN1_DATA".SISTEM_BASLADI;
      A(;
      L     "AI-SENSOR-DATA".JEN1_IC_SICAKLIK_ANLIK;
      L     "JEN1_DATA".SICAKLIK_SET_POINT_2;
      >=R;
      );
      O     "JEN1_DATA".SICAKLIK_SET2_OK;
      );
      =     L 2.0;
      A     L 2.0;
      BLD   102;
      =     "JEN1_DATA".SICAKLIK_SET2_OK;
      A     L 2.0;
      FP    M 754.4;
      JNB   _007;
      L     4;
      T     "JEN1_DATA".STATUS;
_007: NOP   0;
NETWORK
TITLE =
      A     "OTOMATIK";
      A(;
      L     "JEN1_DATA".FAZ_GECISI_STATUS;
      L     1;
      ==I;
      );
      AN    "JEN1_DATA".STOP_SET_RESET;
      A(;
      O(;
      L     "AI-SENSOR-DATA".JEN1_BASINC_ANLIK;
      L     4.600000e+00;
      >R;
      );
      O     "JEN1_DATA".BAR_5_E_ULASTI;
      );
      =     "JEN1_DATA".BAR_5_E_ULASTI;
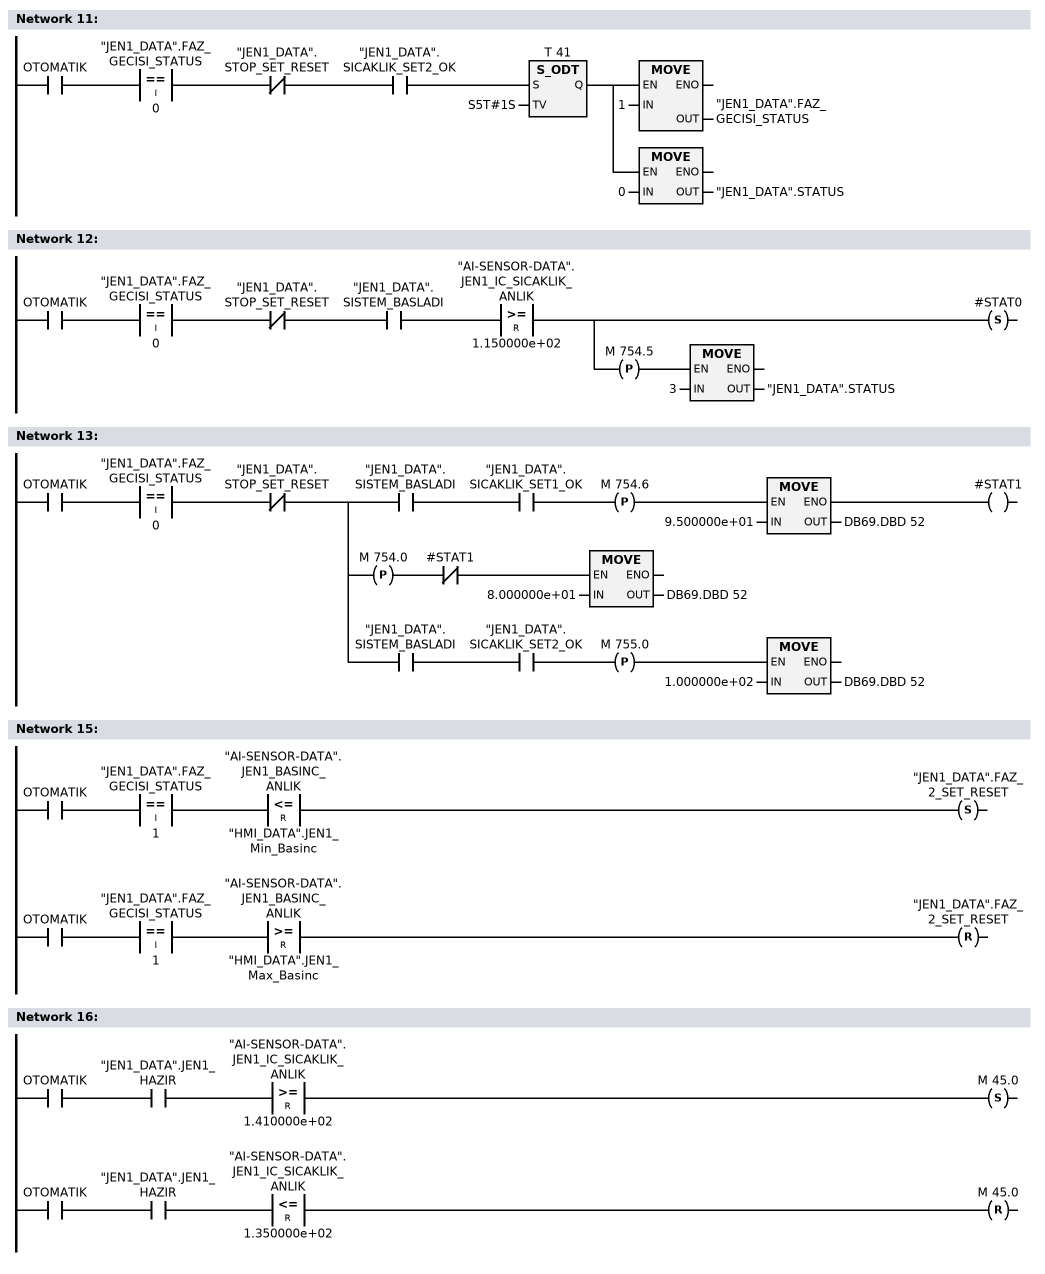
NETWORK
TITLE =
      A     "OTOMATIK";
      A(;
      L     "JEN1_DATA".FAZ_GECISI_STATUS;
      L     0;
      ==I;
      );
      AN    "JEN1_DATA".STOP_SET_RESET;
      A     "JEN1_DATA".SICAKLIK_SET2_OK;
      L     S5T#1S;
      SD    T 41;
      NOP   0;
      NOP   0;
      NOP   0;
      A     T 41;
      =     L 2.0;
      A     L 2.0;
      JNB   _008;
      L     1;
      T     "JEN1_DATA".FAZ_GECISI_STATUS;
_008: NOP   0;
      A     L 2.0;
      JNB   _009;
      L     0;
      T     "JEN1_DATA".STATUS;
_009: NOP   0;
NETWORK
TITLE =
      A     "OTOMATIK";
      A(;
      L     "JEN1_DATA".FAZ_GECISI_STATUS;
      L     0;
      ==I;
      );
      AN    "JEN1_DATA".STOP_SET_RESET;
      A     "JEN1_DATA".SISTEM_BASLADI;
      A(;
      L     "AI-SENSOR-DATA".JEN1_IC_SICAKLIK_ANLIK;
      L     1.150000e+02;
      >=R;
      );
      =     L 2.0;
      A     L 2.0;
      BLD   102;
      S     #STAT0;
      A     L 2.0;
      FP    M 754.5;
      JNB   _00a;
      L     3;
      T     "JEN1_DATA".STATUS;
_00a: NOP   0;
NETWORK
TITLE =
      A     "OTOMATIK";
      A(;
      L     "JEN1_DATA".FAZ_GECISI_STATUS;
      L     0;
      ==I;
      );
      AN    "JEN1_DATA".STOP_SET_RESET;
      =     L 2.0;
      A     L 2.0;
      A     "JEN1_DATA".SISTEM_BASLADI;
      A     "JEN1_DATA".SICAKLIK_SET1_OK;
      FP    M 754.6;
      JNB   _00b;
      L     9.500000e+01;
      T     DB69.DBD 52;
      SET;
      SAVE;
      CLR;
_00b: A     BR;
      =     #STAT1;
      A     L 2.0;
      FP    M 754.0;
      AN    #STAT1;
      JNB   _00c;
      L     8.000000e+01;
      T     DB69.DBD 52;
_00c: NOP   0;
      A     L 2.0;
      A     "JEN1_DATA".SISTEM_BASLADI;
      A     "JEN1_DATA".SICAKLIK_SET2_OK;
      FP    M 755.0;
      JNB   _00d;
      L     1.000000e+02;
      T     DB69.DBD 52;
_00d: NOP   0;
NETWORK
TITLE =
NETWORK
TITLE =
      A     "OTOMATIK";
      A(;
      L     "JEN1_DATA".FAZ_GECISI_STATUS;
      L     1;
      ==I;
      );
      A(;
      L     "AI-SENSOR-DATA".JEN1_BASINC_ANLIK;
      L     "HMI_DATA".JEN1_Min_Basinc;
      <=R;
      );
      S     "JEN1_DATA".FAZ_2_SET_RESET;
      A     "OTOMATIK";
      A(;
      L     "JEN1_DATA".FAZ_GECISI_STATUS;
      L     1;
      ==I;
      );
      A(;
      L     "AI-SENSOR-DATA".JEN1_BASINC_ANLIK;
      L     "HMI_DATA".JEN1_Max_Basinc;
      >=R;
      );
      R     "JEN1_DATA".FAZ_2_SET_RESET;
      NOP   0;
NETWORK
TITLE =
      A     "OTOMATIK";
      A     "JEN1_DATA".JEN1_HAZIR;
      A(;
      L     "AI-SENSOR-DATA".JEN1_IC_SICAKLIK_ANLIK;
      L     1.410000e+02;
      >=R;
      );
      S     M 45.0;
      A     "OTOMATIK";
      A     "JEN1_DATA".JEN1_HAZIR;
      A(;
      L     "AI-SENSOR-DATA".JEN1_IC_SICAKLIK_ANLIK;
      L     1.350000e+02;
      <=R;
      );
      R     M 45.0;
      NOP   0;
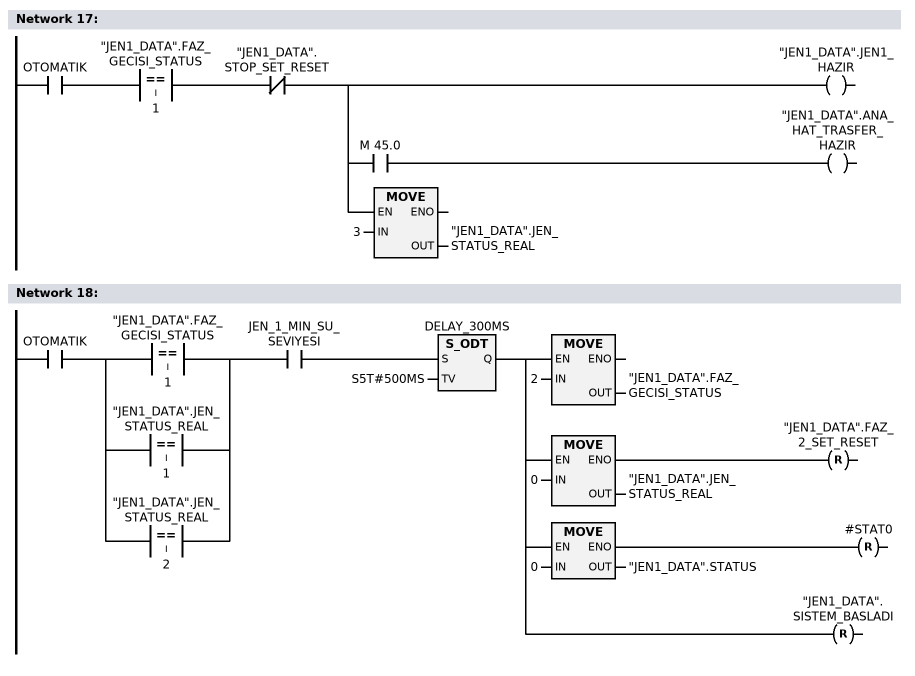
NETWORK
TITLE =
      A     "OTOMATIK";
      A(;
      L     "JEN1_DATA".FAZ_GECISI_STATUS;
      L     1;
      ==I;
      );
      AN    "JEN1_DATA".STOP_SET_RESET;
      =     L 2.0;
      A     L 2.0;
      BLD   102;
      =     "JEN1_DATA".JEN1_HAZIR;
      A     L 2.0;
      A     M 45.0;
      =     "JEN1_DATA".ANA_HAT_TRASFER_HAZIR;
      A     L 2.0;
      JNB   _00e;
      L     3;
      T     "JEN1_DATA".JEN_STATUS_REAL;
_00e: NOP   0;
NETWORK
TITLE =
      A     "OTOMATIK";
      A(;
      O(;
      L     "JEN1_DATA".FAZ_GECISI_STATUS;
      L     1;
      ==I;
      );
      O(;
      L     "JEN1_DATA".JEN_STATUS_REAL;
      L     1;
      ==I;
      );
      O(;
      L     "JEN1_DATA".JEN_STATUS_REAL;
      L     2;
      ==I;
      );
      );
      A     "JEN_1_MIN_SU_SEVIYESI";
      L     S5T#500MS;
      SD    "DELAY_300MS";
      NOP   0;
      NOP   0;
      NOP   0;
      A     "DELAY_300MS";
      =     L 2.0;
      A     L 2.0;
      JNB   _00f;
      L     2;
      T     "JEN1_DATA".FAZ_GECISI_STATUS;
_00f: NOP   0;
      A     L 2.0;
      JNB   _010;
      L     0;
      T     "JEN1_DATA".JEN_STATUS_REAL;
      SET;
      SAVE;
      CLR;
_010: A     BR;
      R     "JEN1_DATA".FAZ_2_SET_RESET;
      A     L 2.0;
      JNB   _011;
      L     0;
      T     "JEN1_DATA".STATUS;
      SET;
      SAVE;
      CLR;
_011: A     BR;
      R     #STAT0;
      A     L 2.0;
      BLD   102;
      R     "JEN1_DATA".SISTEM_BASLADI;
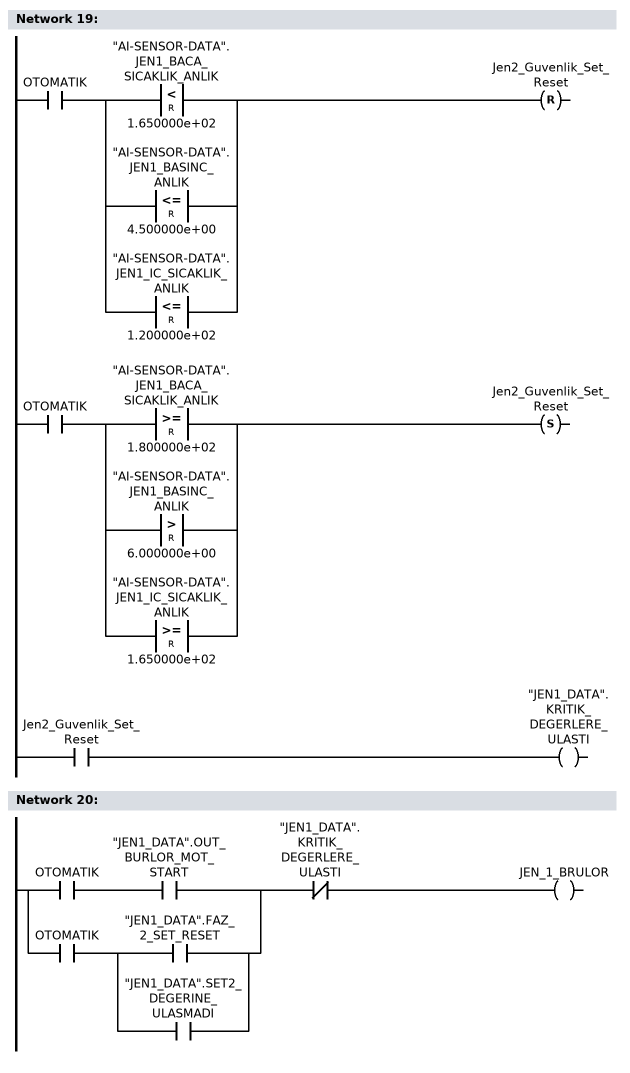
NETWORK
TITLE =
      A     "OTOMATIK";
      A(;
      O(;
      L     "AI-SENSOR-DATA".JEN1_BACA_SICAKLIK_ANLIK;
      L     1.650000e+02;
      <R;
      );
      O(;
      L     "AI-SENSOR-DATA".JEN1_BASINC_ANLIK;
      L     4.500000e+00;
      <=R;
      );
      O(;
      L     "AI-SENSOR-DATA".JEN1_IC_SICAKLIK_ANLIK;
      L     1.200000e+02;
      <=R;
      );
      );
      R     "Jen2_Guvenlik_Set_Reset";
      A     "OTOMATIK";
      A(;
      O(;
      L     "AI-SENSOR-DATA".JEN1_BACA_SICAKLIK_ANLIK;
      L     1.800000e+02;
      >=R;
      );
      O(;
      L     "AI-SENSOR-DATA".JEN1_BASINC_ANLIK;
      L     6.000000e+00;
      >R;
      );
      O(;
      L     "AI-SENSOR-DATA".JEN1_IC_SICAKLIK_ANLIK;
      L     1.650000e+02;
      >=R;
      );
      );
      S     "Jen2_Guvenlik_Set_Reset";
      A     "Jen2_Guvenlik_Set_Reset";
      =     "JEN1_DATA".KRITIK_DEGERLERE_ULASTI;
NETWORK
TITLE =
      A(;
      A     "OTOMATIK";
      A     "JEN1_DATA".OUT_BURLOR_MOT_START;
      O;
      A     "OTOMATIK";
      A(;
      O     "JEN1_DATA".FAZ_2_SET_RESET;
      O     "JEN1_DATA".SET2_DEGERINE_ULASMADI;
      );
      );
      AN    "JEN1_DATA".KRITIK_DEGERLERE_ULASTI;
      =     "JEN_1_BRULOR";
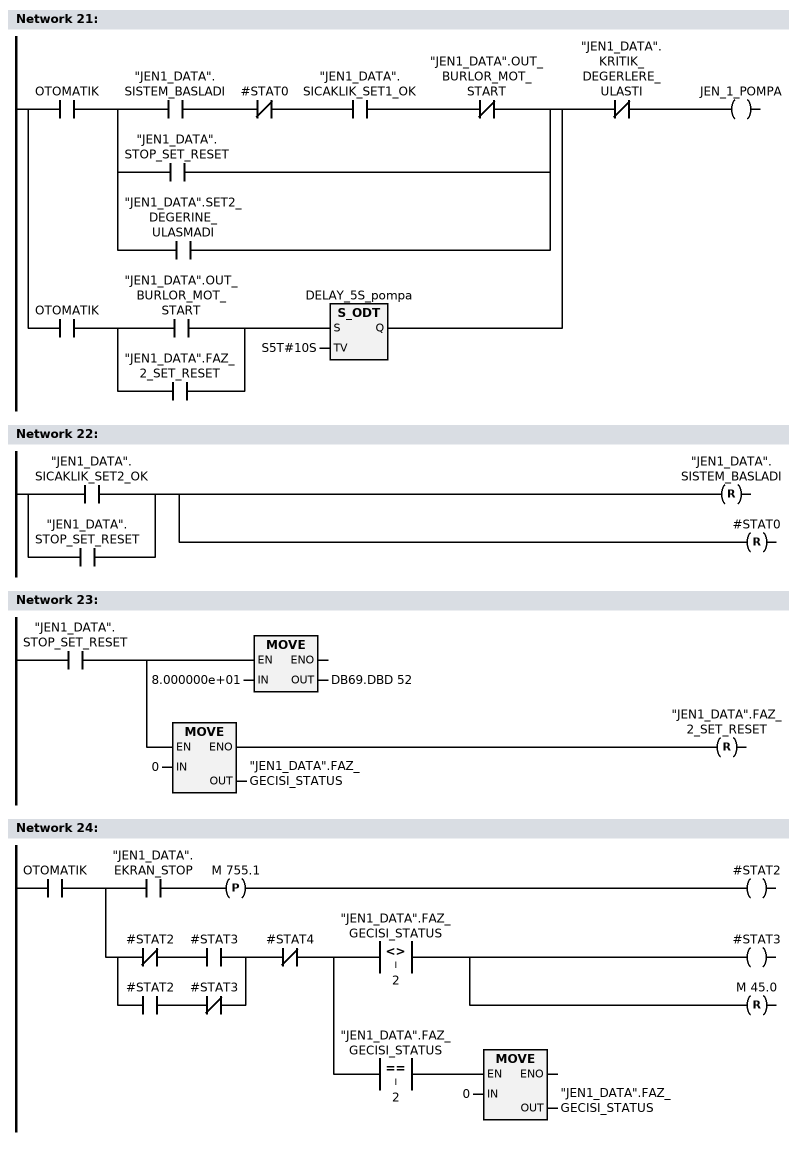
NETWORK
TITLE =
      A(;
      A     "OTOMATIK";
      A(;
      A     "JEN1_DATA".SISTEM_BASLADI;
      AN    #STAT0;
      A     "JEN1_DATA".SICAKLIK_SET1_OK;
      AN    "JEN1_DATA".OUT_BURLOR_MOT_START;
      O     "JEN1_DATA".STOP_SET_RESET;
      O     "JEN1_DATA".SET2_DEGERINE_ULASMADI;
      );
      O(;
      A     "OTOMATIK";
      A(;
      O     "JEN1_DATA".OUT_BURLOR_MOT_START;
      O     "JEN1_DATA".FAZ_2_SET_RESET;
      );
      L     S5T#10S;
      SD    "DELAY_5S_pompa";
      NOP   0;
      NOP   0;
      NOP   0;
      A     "DELAY_5S_pompa";
      );
      );
      AN    "JEN1_DATA".KRITIK_DEGERLERE_ULASTI;
      =     "JEN_1_POMPA";
NETWORK
TITLE =
      O     "JEN1_DATA".SICAKLIK_SET2_OK;
      O     "JEN1_DATA".STOP_SET_RESET;
      R     "JEN1_DATA".SISTEM_BASLADI;
      R     #STAT0;
NETWORK
TITLE =
      A     "JEN1_DATA".STOP_SET_RESET;
      =     L 2.0;
      A     L 2.0;
      JNB   _012;
      L     8.000000e+01;
      T     DB69.DBD 52;
_012: NOP   0;
      A     L 2.0;
      JNB   _013;
      L     0;
      T     "JEN1_DATA".FAZ_GECISI_STATUS;
      SET;
      SAVE;
      CLR;
_013: A     BR;
      R     "JEN1_DATA".FAZ_2_SET_RESET;
NETWORK
TITLE =
      A     "OTOMATIK";
      =     L 2.0;
      A     L 2.0;
      A     "JEN1_DATA".EKRAN_STOP;
      FP    M 755.1;
      =     #STAT2;
      A     L 2.0;
      A(;
      AN    #STAT2;
      A     #STAT3;
      O;
      A     #STAT2;
      AN    #STAT3;
      );
      AN    #STAT4;
      =     L 2.1;
      A     L 2.1;
      A(;
      L     "JEN1_DATA".FAZ_GECISI_STATUS;
      L     2;
      <>I;
      );
      =     #STAT3;
      R     M 45.0;
      A     L 2.1;
      A(;
      L     "JEN1_DATA".FAZ_GECISI_STATUS;
      L     2;
      ==I;
      );
      JNB   _014;
      L     0;
      T     "JEN1_DATA".FAZ_GECISI_STATUS;
_014: NOP   0;
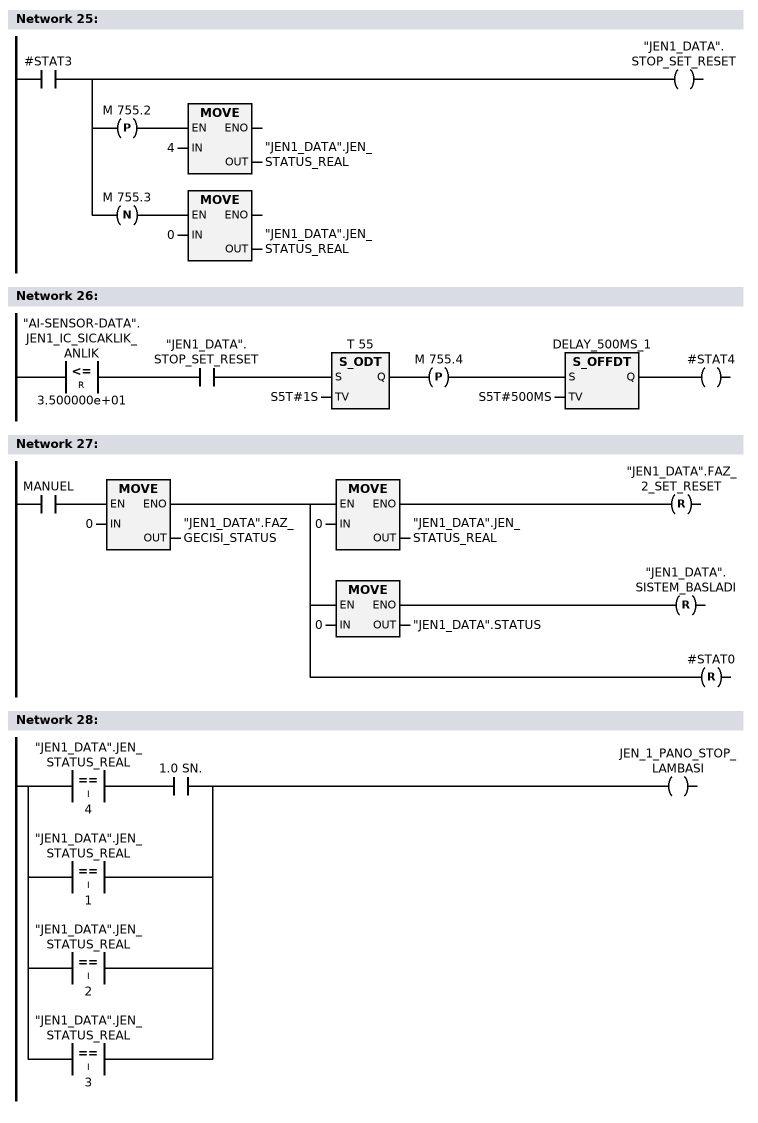
NETWORK
TITLE =
      A     #STAT3;
      =     L 2.0;
      A     L 2.0;
      BLD   102;
      =     "JEN1_DATA".STOP_SET_RESET;
      A     L 2.0;
      FP    M 755.2;
      JNB   _015;
      L     4;
      T     "JEN1_DATA".JEN_STATUS_REAL;
_015: NOP   0;
      A     L 2.0;
      FN    M 755.3;
      JNB   _016;
      L     0;
      T     "JEN1_DATA".JEN_STATUS_REAL;
_016: NOP   0;
NETWORK
TITLE =
      A(;
      A(;
      L     "AI-SENSOR-DATA".JEN1_IC_SICAKLIK_ANLIK;
      L     3.500000e+01;
      <=R;
      );
      A     "JEN1_DATA".STOP_SET_RESET;
      L     S5T#1S;
      SD    T 55;
      NOP   0;
      NOP   0;
      NOP   0;
      A     T 55;
      );
      FP    M 755.4;
      L     S5T#500MS;
      SF    "DELAY_500MS_1";
      NOP   0;
      NOP   0;
      NOP   0;
      A     "DELAY_500MS_1";
      =     #STAT4;
NETWORK
TITLE =
      A     "MANUEL";
      JNB   _017;
      L     0;
      T     "JEN1_DATA".FAZ_GECISI_STATUS;
      SET;
      SAVE;
      CLR;
_017: A     BR;
      =     L 2.0;
      A     L 2.0;
      JNB   _018;
      L     0;
      T     "JEN1_DATA".JEN_STATUS_REAL;
      SET;
      SAVE;
      CLR;
_018: A     BR;
      R     "JEN1_DATA".FAZ_2_SET_RESET;
      A     L 2.0;
      JNB   _019;
      L     0;
      T     "JEN1_DATA".STATUS;
      SET;
      SAVE;
      CLR;
_019: A     BR;
      R     "JEN1_DATA".SISTEM_BASLADI;
      A     L 2.0;
      BLD   102;
      R     #STAT0;
NETWORK
TITLE =
      A(;
      L     "JEN1_DATA".JEN_STATUS_REAL;
      L     4;
      ==I;
      );
      A     "1.0 SN.";
      O(;
      L     "JEN1_DATA".JEN_STATUS_REAL;
      L     1;
      ==I;
      );
      O(;
      L     "JEN1_DATA".JEN_STATUS_REAL;
      L     2;
      ==I;
      );
      O(;
      L     "JEN1_DATA".JEN_STATUS_REAL;
      L     3;
      ==I;
      );
      =     "JEN_1_PANO_STOP_LAMBASI";
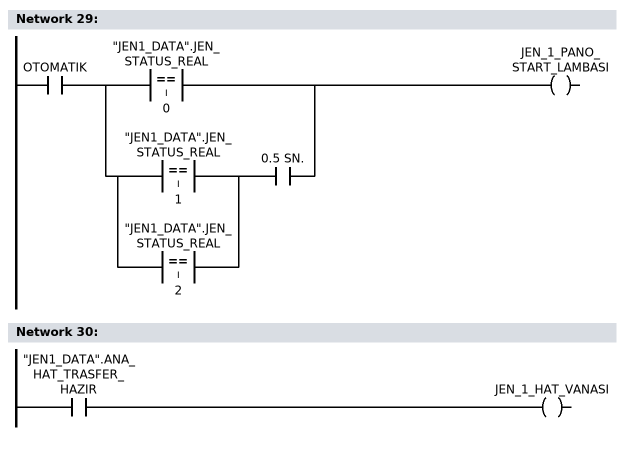
NETWORK
TITLE =
      A     "OTOMATIK";
      A(;
      O(;
      L     "JEN1_DATA".JEN_STATUS_REAL;
      L     0;
      ==I;
      );
      O;
      A(;
      O(;
      L     "JEN1_DATA".JEN_STATUS_REAL;
      L     1;
      ==I;
      );
      O(;
      L     "JEN1_DATA".JEN_STATUS_REAL;
      L     2;
      ==I;
      );
      );
      A     "0.5 SN.";
      );
      =     "JEN_1_PANO_START_LAMBASI";
NETWORK
TITLE =
      A     "JEN1_DATA".ANA_HAT_TRASFER_HAZIR;
      =     "JEN_1_HAT_VANASI";
END_FUNCTION_BLOCK

FUNCTION_BLOCK "JEN2_KONTROL_BLOGU"	// FB 99
VERSION : 0.1
VAR
  STAT0 : BOOL ;
  STAT1 : BOOL ;
  STAT2 : BOOL ;
  STAT3 : BOOL ;
  STAT4 : BOOL ;
  STAT5 : BOOL ;
  STAT6 : BOOL ;
  STAT7 : BOOL ;
  STAT8 : BOOL ;
  STAT9 : BOOL ;
END_VAR
BEGIN
NETWORK
TITLE =
      A     "ALWAYS OFF";
      =     L 0.0;
      BLD   103;
      A(;
      A     "ALWAYS OFF";
      =     L 0.1;
      BLD   103;
      CALL  "SCALE" (
           $1                       := P#P 286.0,
           $2                       := L#1092616192,
           $3                       := L#0,
           $4                       := L 0.1,
           $5                       := "AI-SENSOR-DATA".JEN2_BASINC_RET_VAL,
           $6                       := "AI-SENSOR-DATA".JEN2_BASINC_ANLIK);
      A     BR;
      );
      JNB   _001;
      CALL  "SCALE" (
           $1                       := P#P 288.0,
           $2                       := L#1128792064,
           $3                       := L#0,
           $4                       := L 0.0,
           $5                       := "AI-SENSOR-DATA".JEN2_IC_SICAKLIK_RET_VAL,
           $6                       := "AI-SENSOR-DATA".JEN2_IC_SICAKLIK_ANLIK);
_001: NOP   0;
